ABB RobotStudio station: Cell1234 280921_GPA546_A0610_publ2.rspag

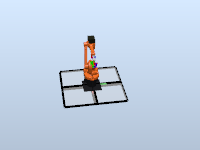
--- station ---
Station Cell1234 pubV2 (saved by RobotStudio 21.2.9526.0)
Controller 05-500633_Cell1, task T_PRINCIP: task frame (RAPID world) sits at (0, 0, 393.01) mm in the station
Controller 05-500633_Cell1
  mechanical unit ROB_1: IRB1600_5_145__01_2, 6 joints, base frame (0, 0, 0) mm
Layout (positions relative to the parent item):
  - Pince [mechanism, from Libraries\Pince.rslib] at (451.32, -3.6, 1437.47) mm, rotated rx 176.02 ry -40.72 rz 6.49 deg; joint values [0.0086] (rad or m)
  - BaseRobot [part, from Libraries\BaseRobot.rslib] at (0, 0, 38.61) mm, rotated rx 90 ry 0 rz 90 deg
  - BoitePince [part, from Libraries\BoitePince.rslib] at (-322.09, -37.25, -99.49) mm, rotated rx 0.01 ry 0.17 rz 1.48 deg
  - LogicGate [smart component, from Libraries\LogicGate.rslib]
      properties: Operator=AND; Delay=0
  - LogicGate [smart component, from Libraries\LogicGate.rslib]
      properties: Operator=NOT; Delay=0
  - IRB1600_5_145__01_2 [mechanism, from Robots\IRB1600_5_145__01.rslib] at (0, 0, 393.01) mm; joint values [-0.0095, -0.5091, 0.516, 0.0144, 0.8505, -1.6733] (rad or m)
  - Cellule_1_Composantes [graphiccomponentgroup]
    - 1_Bloc1 [part, from Libraries\Bloc1.rslib] at (-359.6, 653.4, 807.5) mm, rotated rx 126 ry 0 rz 95.5 deg
    - 1_Bloc2 [part, from Libraries\Bloc1.rslib] at (-359.6, 653.4, 807.5) mm, rotated rx 126 ry 0 rz 95.5 deg
    - 1_Bloc3 [part, from Libraries\Bloc3.rslib] at (-359.6, 653.4, 807.5) mm, rotated rx 126 ry 0 rz 95.5 deg
    - 1_Bloc4 [part, from Libraries\Bloc1.rslib] at (-359.6, 653.4, 807.5) mm, rotated rx 126 ry 0 rz 95.5 deg
    - 1_Bloc5 [part, from Libraries\Bloc1.rslib] at (-359.6, 653.4, 807.5) mm, rotated rx 126 ry 0 rz 95.5 deg
    - 1_Bloc6 [part, from Libraries\Bloc1.rslib] at (-359.6, 653.4, 807.5) mm, rotated rx 126 ry 0 rz 95.5 deg
    - 1_Bloc7 [part, from Libraries\Bloc1.rslib] at (-359.6, 653.4, 807.5) mm, rotated rx 126 ry 0 rz 95.5 deg
    - 1_Bloc8 [part, from Libraries\Bloc1.rslib] at (-359.6, 653.4, 807.5) mm, rotated rx 126 ry 0 rz 95.5 deg
    - 1_Bloc9 [part, from Libraries\Bloc1.rslib] at (-359.6, 653.4, 807.5) mm, rotated rx 126 ry 0 rz 95.5 deg
    - 1_Bloc10 [part, from Libraries\Bloc1.rslib] at (-359.6, 653.4, 807.5) mm, rotated rx 126 ry 0 rz 95.5 deg
    - 1_Crayon [part, from Libraries\Crayon.rslib] at (-244.5, 1025, 746) mm, rotated rx 180 ry 0 rz 0 deg
    - 1_Feuille8.5x11 [part, from Libraries\Feuille8.5x11.rslib] at (50, 800, 746.18) mm, rotated rx 0 ry 0 rz 30 deg
    - 1_Glissoire [part, from Libraries\Glissoire.rslib] at (-578.28, 671.48, 751.2) mm, rotated rx 0 ry 0 rz 5.91 deg
    - 1_PorteCrayon [part, from Libraries\PorteCrayon.rslib] at (-244.76, 1025.26, 745.91) mm
    - 1_Table [part, from Libraries\Table.rslib] at (-567.99, 565.9, -5.81) mm, rotated rx 0 ry 0 rz 5.91 deg
    - 1_Piston [mechanism, from Libraries\Piston.rslib] at (-578.34, 672.08, 752) mm, rotated rx 0 ry 0 rz 5.91 deg; joint values [0] (rad or m)
  - Cellule_2_Composantes [graphiccomponentgroup] at (0, 0, 0) mm
    - 2_Crayon [part, from Libraries\Crayon.rslib] at (-467.39, -707.37, 733.8) mm, rotated rx 179.84 ry -1.57 rz -98.83 deg
    - 2_Feuille8.5x11 [part, from Libraries\Feuille8.5x11.rslib] at (-232.98, -884.29, 745.95) mm, rotated rx -0.47 ry -0.18 rz -45.11 deg
    - 2_PorteCrayon [part, from Libraries\PorteCrayon.rslib] at (-467.32, -707.23, 738.97) mm, rotated rx -0.13 ry -1.57 rz -98.83 deg
    - 2_Table [part, from Libraries\Table.rslib] at (-872.9, -1097.81, -9.38) mm, rotated rx -0.48 ry 0.14 rz -7.29 deg
    - 2_Piston [mechanism, from Libraries\Piston.rslib] at (-862.29, -990.75, 748.42) mm, rotated rx -0.48 ry 0.15 rz -6.57 deg; joint values [0] (rad or m)
    - 2_Bloc1 [part, from Libraries\Bloc1.rslib] at (-652.89, -1053.85, 803.97) mm, rotated rx 126.28 ry 0.71 rz 83.59 deg
    - 2_Bloc2 [part, from Libraries\Bloc1.rslib] at (-652.89, -1053.85, 803.97) mm, rotated rx 126.28 ry 0.71 rz 83.89 deg
    - 2_Bloc3 [part, from Libraries\Bloc3.rslib] at (-652.89, -1053.85, 803.97) mm, rotated rx 126.28 ry 0.71 rz 83.59 deg
    - 2_Bloc4 [part, from Libraries\Bloc1.rslib] at (-652.89, -1053.85, 803.97) mm, rotated rx 126.28 ry 0.71 rz 83.59 deg
    - 2_Bloc5 [part, from Libraries\Bloc1.rslib] at (-652.89, -1053.85, 803.97) mm, rotated rx 126.28 ry 0.71 rz 83.59 deg
    - 2_Bloc6 [part, from Libraries\Bloc1.rslib] at (-652.89, -1053.85, 803.97) mm, rotated rx 126.28 ry 0.71 rz 83.59 deg
    - 2_Bloc7 [part, from Libraries\Bloc1.rslib] at (-652.89, -1053.85, 803.97) mm, rotated rx 126.28 ry 0.71 rz 83.59 deg
    - 2_Bloc8 [part, from Libraries\Bloc1.rslib] at (-652.89, -1053.85, 803.97) mm, rotated rx 126.28 ry 0.71 rz 83.59 deg
    - 2_Bloc9 [part, from Libraries\Bloc1.rslib] at (-652.89, -1053.85, 803.97) mm, rotated rx 126.28 ry 0.71 rz 83.59 deg
    - 2_Bloc10 [part, from Libraries\Bloc1.rslib] at (-652.89, -1053.85, 803.97) mm, rotated rx 126.28 ry 0.71 rz 83.59 deg
    - 2_Glissoire [part, from Libraries\Glissoire.rslib] at (-862.4, -991.66, 747.63) mm, rotated rx -0.48 ry 0.15 rz -6.57 deg
  - Cellule_4_Composantes [graphiccomponentgroup]
    - 4_Bloc1 [part, from Libraries\Bloc1.rslib] at (63.43, -1118.07, 750.5) mm, rotated rx 125.72 ry -2.22 rz 111.85 deg
    - 4_Bloc2 [part, from Libraries\Bloc1.rslib] at (63.43, -1118.07, 750.5) mm, rotated rx 125.72 ry -2.22 rz 111.85 deg
    - 4_Bloc3 [part, from Libraries\Bloc3.rslib] at (63.43, -1118.07, 750.5) mm, rotated rx 125.72 ry -2.22 rz 111.85 deg
    - 4_Bloc4 [part, from Libraries\Bloc1.rslib] at (63.43, -1118.07, 750.5) mm, rotated rx 125.72 ry -2.22 rz 111.85 deg
    - 4_Bloc5 [part, from Libraries\Bloc1.rslib] at (63.43, -1118.07, 750.5) mm, rotated rx 125.72 ry -2.22 rz 111.85 deg
    - 4_Bloc6 [part, from Libraries\Bloc1.rslib] at (63.43, -1118.07, 750.5) mm, rotated rx 125.72 ry -2.22 rz 111.85 deg
    - 4_Bloc7 [part, from Libraries\Bloc1.rslib] at (63.43, -1118.07, 750.5) mm, rotated rx 125.72 ry -2.22 rz 111.85 deg
    - 4_Bloc8 [part, from Libraries\Bloc1.rslib] at (63.43, -1118.07, 750.5) mm, rotated rx 125.72 ry -2.22 rz 111.85 deg
    - 4_Bloc9 [part, from Libraries\Bloc1.rslib] at (63.43, -1118.07, 750.5) mm, rotated rx 125.72 ry -2.22 rz 111.85 deg
    - 4_Bloc10 [part, from Libraries\Bloc1.rslib] at (63.43, -1118.07, 750.5) mm, rotated rx 125.72 ry -2.22 rz 111.85 deg
    - 4_Crayon [part, from Libraries\Crayon.rslib] at (94.76, -713.92, 704.73) mm, rotated rx 177.67 ry 0.01 rz -158.51 deg
    - 4_Feuille8.5x11 [part, from Libraries\Feuille8.5x11.rslib] at (445.38, -893.28, 690.04) mm, rotated rx 2.33 ry -0.01 rz 21.49 deg
    - 4_PorteCrayon [part, from Libraries\PorteCrayon.rslib] at (94.76, -713.92, 704.73) mm, rotated rx 2.33 ry -0.01 rz 21.49 deg
    - 4_Glissoire [part, from Libraries\Glissoire.rslib] at (-151.57, -1158.7, 694.69) mm, rotated rx 2.33 ry -0.01 rz 21.49 deg
    - 4_Table [part, from Libraries\Table.rslib] at (-113.25, -1225.41, -65.44) mm, rotated rx 2.33 ry -0.01 rz 21.49 deg
    - 4_Piston [mechanism, from Libraries\Piston.rslib] at (-151.91, -1157.85, 695.52) mm, rotated rx 2.33 ry -0.01 rz 21.49 deg; joint values [0] (rad or m)
  - Cellule_3_Composantes [graphiccomponentgroup]
    - 3_Bloc1 [part, from Libraries\Bloc1.rslib] at (-255.93, 676.35, 796.95) mm, rotated rx 125.68 ry -0.79 rz 86.11 deg
    - 3_Bloc2 [part, from Libraries\Bloc1.rslib] at (-255.93, 676.35, 796.95) mm, rotated rx 125.68 ry -0.79 rz 86.11 deg
    - 3_Bloc3 [part, from Libraries\Bloc3.rslib] at (-255.93, 676.35, 796.95) mm, rotated rx 125.68 ry -0.79 rz 86.11 deg
    - 3_Bloc4 [part, from Libraries\Bloc1.rslib] at (-255.93, 676.35, 796.95) mm, rotated rx 125.68 ry -0.79 rz 86.11 deg
    - 3_Bloc5 [part, from Libraries\Bloc1.rslib] at (-255.93, 676.35, 796.95) mm, rotated rx 125.68 ry -0.79 rz 86.11 deg
    - 3_Bloc6 [part, from Libraries\Bloc1.rslib] at (-255.93, 676.35, 796.95) mm, rotated rx 125.68 ry -0.79 rz 86.11 deg
    - 3_Bloc7 [part, from Libraries\Bloc1.rslib] at (-255.93, 676.35, 796.95) mm, rotated rx 125.68 ry -0.79 rz 86.11 deg
    - 3_Bloc8 [part, from Libraries\Bloc1.rslib] at (-255.93, 676.35, 796.95) mm, rotated rx 125.68 ry -0.79 rz 86.11 deg
    - 3_Bloc9 [part, from Libraries\Bloc1.rslib] at (-255.93, 676.35, 796.95) mm, rotated rx 126.68 ry -0.79 rz 86.11 deg
    - 3_Bloc10 [part, from Libraries\Bloc1.rslib] at (-255.93, 676.35, 796.95) mm, rotated rx 125.68 ry -0.79 rz 86.11 deg
    - 3_Crayon [part, from Libraries\Crayon.rslib] at (-66.31, 1010.69, 738.78) mm, rotated rx -179.88 ry 1.4 rz -95.14 deg
    - 3_Feuille8.5x11 [part, from Libraries\Feuille8.5x11.rslib] at (52.4, 669.01, 746.18) mm, rotated rx 0 ry 0 rz 1.76 deg
    - 3_Glissoire [part, from Libraries\Glissoire.rslib] at (-467.56, 729.54, 741.03) mm, rotated rx 0.36 ry 0.24 rz -3.84 deg
    - 3_PorteCrayon [part, from Libraries\PorteCrayon.rslib] at (-66.84, 1007.76, 860.12) mm, rotated rx -179.88 ry 1.4 rz -95.14 deg
    - 3_Table [part, from Libraries\Table.rslib] at (-484.28, 629.79, -18.55) mm, rotated rx 0.28 ry 0 rz -5.2 deg
    - 3_Piston [mechanism, from Libraries\Piston.rslib] at (-467.45, 731.2, 741.83) mm, rotated rx 0.36 ry 0.24 rz -3.84 deg; joint values [0] (rad or m)
Attachment: 1_PorteCrayon is attached to 1_Table
Attachment: 1_Piston is attached to 1_Glissoire
Attachment: Pince is attached to IRB1600_5_145__01_2 / Link6
Attachment: BoitePince is attached to IRB1600_5_145__01_2 / Link3
Attachment: 2_PorteCrayon is attached to 2_Table
Attachment: 2_Piston is attached to 2_Glissoire
Attachment: 4_PorteCrayon is attached to 4_Table
Attachment: 4_Piston is attached to 4_Glissoire
Attachment: 3_PorteCrayon is attached to 3_Table
Attachment: 3_Piston is attached to 3_Glissoire
EventTableEntry 2774: Group=, Trigger=DO01_EE_PINCE01 2775, Actions=[EventTableActionAttach 2776], Comment=Attache l'objet le plus proche a la pince, devrait normalement être un bloc quand dans le glissoire ou le crayon, ActivationMode=2, Cyclic=false
EventTableTriggerIO 2775: IOValue=[1], IRC5Controller=? -1, Operator=0, SignalSource=05-500633_Cell1 2885
EventTableActionAttach 2776: AttachmentParent=Pince 925, AttachmentChild=? -1, MountObject=false, Offset=[X=1, Y=0, Z=0, W=0, X=0, Y=1, Z=0, W=0, X=0, Y=0, Z=1, W=0, X=0, Y=0, Z=0, W=1], FlangeIndext=0, FindNearest=true
EventTableTriggerIO 2777: IOValue=[0], IRC5Controller=? -1, Operator=0, SignalSource=05-500633_Cell1 2885
EventTableEntry 2778: Group=, Trigger=DO01_EE_PINCE01 2777, Actions=[EventTableActionDetach 2779], Comment=relache ce que le robot tiens., ActivationMode=2, Cyclic=false
EventTableActionDetach 2779: AttachmentParent=Pince 925, AttachmentChild=? -1
EventTableEntry 2780: Group=, Trigger=INIT_GAUCHE 2781, Actions=[EventTableActionMove 5190, EventTableActionMove 5191, EventTableActionMove 5192, EventTableActionMove 5193, EventTableActionMove 5194, EventTableActionMove 5195, EventTableActionMove 5196, EventTableActionMove 5197, EventTableActionMove 5198, EventTableActionMove 5199, EventTableActionMove 5200, EventTableActionMove 5201, EventTableActionMove 5202, EventTableActionMove 5203, EventTableActionMove 5204, EventTableActionDetach 5205, DO09_FV0101 5206, PistonIN 5207, PistonOUT 5208, DI13_ZS0103 5209, DI09_ZS0101 5210, TrouAGauche 5211, INIT_GAUCHE 5212, INIT_DROITE 5213, EventTableActionMove 5214, EventTableActionMove 5215, EventTableActionMove 5216, EventTableActionMove 5217, EventTableActionMove 5218, EventTableActionMove 5219, EventTableActionMove 5220, EventTableActionMove 5221, EventTableActionMove 5222, EventTableActionMove 5223, EventTableActionMove 5237, EventTableActionMove 5238, EventTableActionMove 5239, EventTableActionMove 5240, EventTableActionMove 5241, EventTableActionMove 5242, EventTableActionMove 5243, EventTableActionMove 5244, EventTableActionMove 5245, EventTableActionMove 5246, EventTableActionMove 5247, EventTableActionMove 5248, EventTableActionMove 5249, EventTableActionMove 5250, EventTableActionMove 5251, EventTableActionMove 5252, EventTableActionMove 5253, EventTableActionMove 5254, EventTableActionMove 5255, EventTableActionMove 5256], Comment=Replace les 10 blocs dans la zone de prise,
replace le glissoire
replace la table
replace la feuille
replace le crayon et sa base
détache ce que la pince peut tenir
place les valeurs du verin, ActivationMode=2, Cyclic=false
EventTableTriggerIO 2781: IOValue=[1], IRC5Controller=? -1, Operator=0, SignalSource=Cell1234 pubV2 1
EventTableEntry 2812: Group=, Trigger=DO01_EE_PINCE01 2813, Actions=[EventTableActionMechanicalPose 2814], Comment=, ActivationMode=2, Cyclic=false
EventTableTriggerIO 2813: IOValue=[1], IRC5Controller=? -1, Operator=0, SignalSource=05-500633_Cell1 2885
EventTableActionMechanicalPose 2814: VirtualSignal=, Mechanism=Pince 925, ToPoseName=Closed, VirtualSignalValue=[1]
EventTableTriggerIO 2815: IOValue=[0], IRC5Controller=? -1, Operator=0, SignalSource=05-500633_Cell1 2885
EventTableEntry 2816: Group=, Trigger=DO01_EE_PINCE01 2815, Actions=[EventTableActionMechanicalPose 2817], Comment=, ActivationMode=2, Cyclic=false
EventTableActionMechanicalPose 2817: VirtualSignal=, Mechanism=Pince 925, ToPoseName=Opened, VirtualSignalValue=[1]
EventTableEntry 2818: Group=, Trigger=DO09_FV0101 2819, Actions=[EventTableActionMechanicalPose 2820, PistonIN 2822], Comment=, ActivationMode=2, Cyclic=false
EventTableTriggerIO 2819: IOValue=[1], IRC5Controller=? -1, Operator=0, SignalSource=05-500633_Cell1 2885
EventTableActionMechanicalPose 2820: VirtualSignal=PistonOUT, Mechanism=1_Piston 921, ToPoseName=OUT, VirtualSignalValue=[1]
EventTableTriggerIO 2821: IOValue=[0], IRC5Controller=? -1, Operator=0, SignalSource=05-500633_Cell1 2885
EventTableActionIO 2822: IOValue=[0], IRC5Controller=? -1, SignalTarget=Cell1234 pubV2 1
EventTableEntry 2823: Group=, Trigger=DO09_FV0101 2821, Actions=[EventTableActionMechanicalPose 2824, PistonOUT 2825], Comment=, ActivationMode=2, Cyclic=false
EventTableActionMechanicalPose 2824: VirtualSignal=PistonIN, Mechanism=1_Piston 921, ToPoseName=IN, VirtualSignalValue=[1]
EventTableActionIO 2825: IOValue=[0], IRC5Controller=? -1, SignalTarget=Cell1234 pubV2 1
EventTableTriggerIO 2847: IOValue=[1], IRC5Controller=? -1, Operator=0, SignalSource=Cell1234 pubV2 1
EventTableEntry 2848: Group=, Trigger=INIT_DROITE 2847, Actions=[EventTableActionMove 5156, EventTableActionMove 5157, EventTableActionMove 5158, EventTableActionMove 5159, EventTableActionMove 5160, EventTableActionMove 5161, EventTableActionMove 5162, EventTableActionMove 5163, EventTableActionMove 5164, EventTableActionMove 5165, EventTableActionMove 5166, EventTableActionMove 5167, EventTableActionMove 5168, EventTableActionMove 5169, EventTableActionMove 5170, EventTableActionDetach 5171, DO09_FV0101 5172, PistonIN 5173, PistonOUT 5174, DI13_ZS0103 5175, DI09_ZS0101 5176, TrouAGauche 5177, INIT_DROITE 5178, INIT_GAUCHE 5179, EventTableActionMove 5180, EventTableActionMove 5181, EventTableActionMove 5182, EventTableActionMove 5183, EventTableActionMove 5184, EventTableActionMove 5185, EventTableActionMove 5186, EventTableActionMove 5187, EventTableActionMove 5188, EventTableActionMove 5189, EventTableActionMove 5224, EventTableActionMove 5225, EventTableActionMove 5226, EventTableActionMove 5227, EventTableActionMove 5228, EventTableActionMove 5232, EventTableActionMove 5233, EventTableActionMove 5234, EventTableActionMove 5235, EventTableActionMove 5236, EventTableActionMove 5257, EventTableActionMove 5258, EventTableActionMove 5259, EventTableActionMove 5260, EventTableActionMove 5261, EventTableActionMove 5262, EventTableActionMove 5263, EventTableActionMove 5264, EventTableActionMove 5265, EventTableActionMove 5266], Comment=Replace les 10 blocs dans la zone de prise,
replace le glissoire
replace la table
replace la feuille
replace le crayon et sa base
détache ce que la pince peut tenir
place les valeurs du verin, ActivationMode=2, Cyclic=false
EventTableTriggerIO 3612: IOValue=[1], IRC5Controller=? -1, Operator=0, SignalSource=05-500633_Cell1 2885
EventTableTriggerIO 3613: IOValue=[0], IRC5Controller=? -1, Operator=0, SignalSource=05-500633_Cell1 2885
EventTableEntry 3614: Group=, Trigger=DO09_FV0101 3612, Actions=[EventTableActionMechanicalPose 3615, PistonIN 3616], Comment=, ActivationMode=2, Cyclic=false
EventTableActionMechanicalPose 3615: VirtualSignal=PistonOUT, Mechanism=2_Piston 3404, ToPoseName=OUT, VirtualSignalValue=[1]
EventTableActionIO 3616: IOValue=[0], IRC5Controller=? -1, SignalTarget=Cell1234 pubV2 1
EventTableEntry 3617: Group=, Trigger=DO09_FV0101 3613, Actions=[EventTableActionMechanicalPose 3618, PistonOUT 3619], Comment=, ActivationMode=2, Cyclic=false
EventTableActionMechanicalPose 3618: VirtualSignal=PistonIN, Mechanism=2_Piston 3404, ToPoseName=IN, VirtualSignalValue=[1]
EventTableActionIO 3619: IOValue=[0], IRC5Controller=? -1, SignalTarget=Cell1234 pubV2 1
EventTableTriggerIO 4329: IOValue=[1], IRC5Controller=? -1, Operator=0, SignalSource=05-500633_Cell1 2885
EventTableTriggerIO 4330: IOValue=[0], IRC5Controller=? -1, Operator=0, SignalSource=05-500633_Cell1 2885
EventTableEntry 4331: Group=, Trigger=DO09_FV0101 4329, Actions=[EventTableActionMechanicalPose 4332, PistonIN 4333], Comment=, ActivationMode=2, Cyclic=false
EventTableActionMechanicalPose 4332: VirtualSignal=PistonOUT, Mechanism=4_Piston 4323, ToPoseName=OUT, VirtualSignalValue=[1]
EventTableActionIO 4333: IOValue=[0], IRC5Controller=? -1, SignalTarget=Cell1234 pubV2 1
EventTableEntry 4334: Group=, Trigger=DO09_FV0101 4330, Actions=[EventTableActionMechanicalPose 4335, PistonOUT 4336], Comment=, ActivationMode=2, Cyclic=false
EventTableActionMechanicalPose 4335: VirtualSignal=PistonIN, Mechanism=4_Piston 4323, ToPoseName=IN, VirtualSignalValue=[1]
EventTableActionIO 4336: IOValue=[0], IRC5Controller=? -1, SignalTarget=Cell1234 pubV2 1
EventTableActionMove 5156: Object=1_Bloc1 943, GlobalTransform=[X=-0.095845752520224, Y=0.995396198367179, Z=0, W=0, X=0.585079205588221, Y=0.0563367198262618, Z=0.809016994374948, W=0, X=0.805292440615264, Y=0.0775408426275167, Z=-0.587785252292473, W=0, X=-0.3596, Y=0.6534, Z=0.8075, W=1]
EventTableActionMove 5157: Object=1_Bloc2 2784, GlobalTransform=[X=-0.095845752520224, Y=0.995396198367179, Z=0, W=0, X=0.585079205588221, Y=0.0563367198262618, Z=0.809016994374948, W=0, X=0.805292440615264, Y=0.0775408426275167, Z=-0.587785252292473, W=0, X=-0.3596, Y=0.6534, Z=0.8075, W=1]
EventTableActionMove 5158: Object=1_Bloc3 942, GlobalTransform=[X=-0.095845752520224, Y=0.995396198367179, Z=0, W=0, X=0.585079205588221, Y=0.0563367198262618, Z=0.809016994374948, W=0, X=0.805292440615264, Y=0.0775408426275167, Z=-0.587785252292473, W=0, X=-0.3596, Y=0.6534, Z=0.8075, W=1]
EventTableActionMove 5159: Object=1_Bloc4 2790, GlobalTransform=[X=-0.095845752520224, Y=0.995396198367179, Z=0, W=0, X=0.585079205588221, Y=0.0563367198262618, Z=0.809016994374948, W=0, X=0.805292440615264, Y=0.0775408426275167, Z=-0.587785252292473, W=0, X=-0.3596, Y=0.6534, Z=0.8075, W=1]
EventTableActionMove 5160: Object=1_Bloc5 2791, GlobalTransform=[X=-0.095845752520224, Y=0.995396198367179, Z=0, W=0, X=0.585079205588221, Y=0.0563367198262618, Z=0.809016994374948, W=0, X=0.805292440615264, Y=0.0775408426275167, Z=-0.587785252292473, W=0, X=-0.3596, Y=0.6534, Z=0.8075, W=1]
EventTableActionMove 5161: Object=1_Bloc6 2792, GlobalTransform=[X=-0.095845752520224, Y=0.995396198367179, Z=0, W=0, X=0.585079205588221, Y=0.0563367198262618, Z=0.809016994374948, W=0, X=0.805292440615264, Y=0.0775408426275167, Z=-0.587785252292473, W=0, X=-0.3596, Y=0.6534, Z=0.8075, W=1]
EventTableActionMove 5162: Object=1_Bloc7 2793, GlobalTransform=[X=-0.095845752520224, Y=0.995396198367179, Z=0, W=0, X=0.585079205588221, Y=0.0563367198262618, Z=0.809016994374948, W=0, X=0.805292440615264, Y=0.0775408426275167, Z=-0.587785252292473, W=0, X=-0.3596, Y=0.6534, Z=0.8075, W=1]
EventTableActionMove 5163: Object=1_Bloc8 2794, GlobalTransform=[X=-0.095845752520224, Y=0.995396198367179, Z=0, W=0, X=0.585079205588221, Y=0.0563367198262618, Z=0.809016994374948, W=0, X=0.805292440615264, Y=0.0775408426275167, Z=-0.587785252292473, W=0, X=-0.3596, Y=0.6534, Z=0.8075, W=1]
EventTableActionMove 5164: Object=1_Bloc9 2795, GlobalTransform=[X=-0.095845752520224, Y=0.995396198367179, Z=0, W=0, X=0.585079205588221, Y=0.0563367198262618, Z=0.809016994374948, W=0, X=0.805292440615264, Y=0.0775408426275167, Z=-0.587785252292473, W=0, X=-0.3596, Y=0.6534, Z=0.8075, W=1]
EventTableActionMove 5165: Object=1_Bloc10 2796, GlobalTransform=[X=-0.095845752520224, Y=0.995396198367179, Z=0, W=0, X=0.585079205588221, Y=0.0563367198262618, Z=0.809016994374948, W=0, X=0.805292440615264, Y=0.0775408426275167, Z=-0.587785252292473, W=0, X=-0.3596, Y=0.6534, Z=0.8075, W=1]
EventTableActionMove 5166: Object=1_Glissoire 932, GlobalTransform=[X=0.994684861284941, Y=0.102966143613121, Z=0, W=0, X=-0.102966143613121, Y=0.994684861284941, Z=0, W=0, X=0, Y=0, Z=1, W=0, X=-0.57828, Y=0.67148, Z=0.751202, W=1]
EventTableActionMove 5167: Object=1_Table 919, GlobalTransform=[X=0.994684861284941, Y=0.102966143613121, Z=0, W=0, X=-0.102966143613121, Y=0.994684861284941, Z=0, W=0, X=0, Y=0, Z=1, W=0, X=-0.567989, Y=0.565905, Z=-0.005814, W=1]
EventTableActionMove 5168: Object=1_Feuille8.5x11 933, GlobalTransform=[X=0.866025403784439, Y=0.5, Z=0, W=0, X=-0.5, Y=0.866025403784439, Z=0, W=0, X=0, Y=0, Z=1, W=0, X=0.05, Y=0.8, Z=0.746181, W=1]
EventTableActionMove 5169: Object=1_PorteCrayon 920, GlobalTransform=[X=1, Y=0, Z=0, W=0, X=0, Y=1, Z=0, W=0, X=0, Y=0, Z=1, W=0, X=-0.244763, Y=1.025263, Z=0.745911, W=1]
EventTableActionMove 5170: Object=1_Crayon 934, GlobalTransform=[X=1, Y=0, Z=0, W=0, X=0, Y=-1, Z=0, W=0, X=0, Y=0, Z=-1, W=0, X=-0.2445, Y=1.025, Z=0.746, W=1]
EventTableActionDetach 5171: AttachmentParent=Pince 925, AttachmentChild=? -1
EventTableActionIO 5172: IOValue=[0], IRC5Controller=? -1, SignalTarget=05-500633_Cell1 2885
EventTableActionIO 5173: IOValue=[1], IRC5Controller=? -1, SignalTarget=Cell1234 pubV2 1
EventTableActionIO 5174: IOValue=[0], IRC5Controller=? -1, SignalTarget=Cell1234 pubV2 1
EventTableActionIO 5175: IOValue=[1], IRC5Controller=? -1, SignalTarget=05-500633_Cell1 2885
EventTableActionIO 5176: IOValue=[1], IRC5Controller=? -1, SignalTarget=05-500633_Cell1 2885
EventTableActionIO 5177: IOValue=[0], IRC5Controller=? -1, SignalTarget=Cell1234 pubV2 1
EventTableActionIO 5178: IOValue=[0], IRC5Controller=? -1, SignalTarget=Cell1234 pubV2 1
EventTableActionIO 5179: IOValue=[0], IRC5Controller=? -1, SignalTarget=Cell1234 pubV2 1
EventTableActionMove 5180: Object=2_Bloc1 3408, GlobalTransform=[X=0.11163380406932, Y=0.993672151168342, Z=-0.0123915205480335, W=0, X=0.589147801205299, Y=-0.0561355574929458, Z=0.806072991434347, W=0, X=0.800276678483119, Y=-0.0972854314758168, Z=-0.591686388806258, W=0, X=-0.65289, Y=-1.05385, Z=0.80397, W=1]
EventTableActionMove 5181: Object=2_Bloc2 3409, GlobalTransform=[X=0.106429442376949, Y=0.994243040716826, Z=-0.0123915205480335, W=0, X=0.589433649061701, Y=-0.0530500314221419, Z=0.806072991434347, W=0, X=0.800775091488952, Y=-0.0930938781675272, Z=-0.591686388806258, W=0, X=-0.65289, Y=-1.05385, Z=0.80397, W=1]
EventTableActionMove 5182: Object=2_Bloc3 3410, GlobalTransform=[X=0.11163380406932, Y=0.993672151168342, Z=-0.0123915205480335, W=0, X=0.589147801205299, Y=-0.0561355574929458, Z=0.806072991434347, W=0, X=0.800276678483119, Y=-0.0972854314758168, Z=-0.591686388806258, W=0, X=-0.65289, Y=-1.05385, Z=0.80397, W=1]
EventTableActionMove 5183: Object=2_Bloc4 3411, GlobalTransform=[X=0.11163380406932, Y=0.993672151168342, Z=-0.0123915205480335, W=0, X=0.589147801205299, Y=-0.0561355574929458, Z=0.806072991434347, W=0, X=0.800276678483119, Y=-0.0972854314758168, Z=-0.591686388806258, W=0, X=-0.65289, Y=-1.05385, Z=0.80397, W=1]
EventTableActionMove 5184: Object=2_Bloc5 3412, GlobalTransform=[X=0.11163380406932, Y=0.993672151168342, Z=-0.0123915205480335, W=0, X=0.589147801205299, Y=-0.0561355574929458, Z=0.806072991434347, W=0, X=0.800276678483119, Y=-0.0972854314758168, Z=-0.591686388806258, W=0, X=-0.65289, Y=-1.05385, Z=0.80397, W=1]
EventTableActionMove 5185: Object=2_Bloc6 3413, GlobalTransform=[X=0.11163380406932, Y=0.993672151168342, Z=-0.0123915205480335, W=0, X=0.589147801205299, Y=-0.0561355574929458, Z=0.806072991434347, W=0, X=0.800276678483119, Y=-0.0972854314758168, Z=-0.591686388806258, W=0, X=-0.65289, Y=-1.05385, Z=0.80397, W=1]
EventTableActionMove 5186: Object=2_Bloc7 3414, GlobalTransform=[X=0.11163380406932, Y=0.993672151168342, Z=-0.0123915205480335, W=0, X=0.589147801205299, Y=-0.0561355574929458, Z=0.806072991434347, W=0, X=0.800276678483119, Y=-0.0972854314758168, Z=-0.591686388806258, W=0, X=-0.65289, Y=-1.05385, Z=0.80397, W=1]
EventTableActionMove 5187: Object=2_Bloc8 3415, GlobalTransform=[X=0.11163380406932, Y=0.993672151168342, Z=-0.0123915205480335, W=0, X=0.589147801205299, Y=-0.0561355574929458, Z=0.806072991434347, W=0, X=0.800276678483119, Y=-0.0972854314758168, Z=-0.591686388806258, W=0, X=-0.65289, Y=-1.05385, Z=0.80397, W=1]
EventTableActionMove 5188: Object=2_Bloc9 3416, GlobalTransform=[X=0.11163380406932, Y=0.993672151168342, Z=-0.0123915205480335, W=0, X=0.589147801205299, Y=-0.0561355574929458, Z=0.806072991434347, W=0, X=0.800276678483119, Y=-0.0972854314758168, Z=-0.591686388806258, W=0, X=-0.65289, Y=-1.05385, Z=0.80397, W=1]
EventTableActionMove 5189: Object=2_Bloc10 3417, GlobalTransform=[X=0.11163380406932, Y=0.993672151168342, Z=-0.0123915205480335, W=0, X=0.589147801205299, Y=-0.0561355574929458, Z=0.806072991434347, W=0, X=0.800276678483119, Y=-0.0972854314758168, Z=-0.591686388806258, W=0, X=-0.65289, Y=-1.05385, Z=0.80397, W=1]
EventTableActionMove 5190: Object=1_Bloc1 943, GlobalTransform=[X=0.0958457525202241, Y=-0.995396198367179, Z=0, W=0, X=-0.815380830769965, Y=-0.0785122441133584, Z=0.573576436351046, W=0, X=-0.570935804216825, Y=-0.0549748651699344, Z=-0.819152044288992, W=0, X=-0.3596, Y=0.6534, Z=0.8075, W=1]
EventTableActionMove 5191: Object=1_Bloc2 2784, GlobalTransform=[X=0.0958457525202241, Y=-0.995396198367179, Z=0, W=0, X=-0.815380830769965, Y=-0.0785122441133584, Z=0.573576436351046, W=0, X=-0.570935804216825, Y=-0.0549748651699344, Z=-0.819152044288992, W=0, X=-0.3596, Y=0.6534, Z=0.8075, W=1]
EventTableActionMove 5192: Object=1_Bloc3 942, GlobalTransform=[X=0.0958457525202241, Y=-0.995396198367179, Z=0, W=0, X=-0.815380830769965, Y=-0.0785122441133584, Z=0.573576436351046, W=0, X=-0.570935804216825, Y=-0.0549748651699344, Z=-0.819152044288992, W=0, X=-0.3596, Y=0.6534, Z=0.8075, W=1]
EventTableActionMove 5193: Object=1_Bloc4 2790, GlobalTransform=[X=0.0958457525202241, Y=-0.995396198367179, Z=0, W=0, X=-0.815380830769965, Y=-0.0785122441133584, Z=0.573576436351046, W=0, X=-0.570935804216825, Y=-0.0549748651699344, Z=-0.819152044288992, W=0, X=-0.3596, Y=0.6534, Z=0.8075, W=1]
EventTableActionMove 5194: Object=1_Bloc5 2791, GlobalTransform=[X=0.0958457525202241, Y=-0.995396198367179, Z=0, W=0, X=-0.815380830769965, Y=-0.0785122441133584, Z=0.573576436351046, W=0, X=-0.570935804216825, Y=-0.0549748651699344, Z=-0.819152044288992, W=0, X=-0.3596, Y=0.6534, Z=0.8075, W=1]
EventTableActionMove 5195: Object=1_Bloc6 2792, GlobalTransform=[X=0.0958457525202241, Y=-0.995396198367179, Z=0, W=0, X=-0.815380830769965, Y=-0.0785122441133584, Z=0.573576436351046, W=0, X=-0.570935804216825, Y=-0.0549748651699344, Z=-0.819152044288992, W=0, X=-0.3596, Y=0.6534, Z=0.8075, W=1]
EventTableActionMove 5196: Object=1_Bloc7 2793, GlobalTransform=[X=0.0958457525202241, Y=-0.995396198367179, Z=0, W=0, X=-0.815380830769965, Y=-0.0785122441133584, Z=0.573576436351046, W=0, X=-0.570935804216825, Y=-0.0549748651699344, Z=-0.819152044288992, W=0, X=-0.3596, Y=0.6534, Z=0.8075, W=1]
EventTableActionMove 5197: Object=1_Bloc8 2794, GlobalTransform=[X=0.0958457525202241, Y=-0.995396198367179, Z=0, W=0, X=-0.815380830769965, Y=-0.0785122441133584, Z=0.573576436351046, W=0, X=-0.570935804216825, Y=-0.0549748651699344, Z=-0.819152044288992, W=0, X=-0.3596, Y=0.6534, Z=0.8075, W=1]
EventTableActionMove 5198: Object=1_Bloc9 2795, GlobalTransform=[X=0.0958457525202241, Y=-0.995396198367179, Z=0, W=0, X=-0.815380830769965, Y=-0.0785122441133584, Z=0.573576436351046, W=0, X=-0.570935804216825, Y=-0.0549748651699344, Z=-0.819152044288992, W=0, X=-0.3596, Y=0.6534, Z=0.8075, W=1]
EventTableActionMove 5199: Object=1_Bloc10 2796, GlobalTransform=[X=0.0958457525202241, Y=-0.995396198367179, Z=0, W=0, X=-0.815380830769965, Y=-0.0785122441133584, Z=0.573576436351046, W=0, X=-0.570935804216825, Y=-0.0549748651699344, Z=-0.819152044288992, W=0, X=-0.3596, Y=0.6534, Z=0.8075, W=1]
EventTableActionMove 5200: Object=1_Glissoire 932, GlobalTransform=[X=0.994684861284941, Y=0.102966143613121, Z=0, W=0, X=-0.102966143613121, Y=0.994684861284941, Z=0, W=0, X=0, Y=0, Z=1, W=0, X=-0.57828, Y=0.67148, Z=0.751202, W=1]
EventTableActionMove 5201: Object=1_Table 919, GlobalTransform=[X=0.994684861284941, Y=0.102966143613121, Z=0, W=0, X=-0.102966143613121, Y=0.994684861284941, Z=0, W=0, X=0, Y=0, Z=1, W=0, X=-0.567989, Y=0.565905, Z=-0.005814, W=1]
EventTableActionMove 5202: Object=1_Feuille8.5x11 933, GlobalTransform=[X=0.866025403784439, Y=0.5, Z=0, W=0, X=-0.5, Y=0.866025403784439, Z=0, W=0, X=0, Y=0, Z=1, W=0, X=0.05, Y=0.8, Z=0.746181, W=1]
EventTableActionMove 5203: Object=1_PorteCrayon 920, GlobalTransform=[X=1, Y=0, Z=0, W=0, X=0, Y=1, Z=0, W=0, X=0, Y=0, Z=1, W=0, X=-0.244763, Y=1.025263, Z=0.745911, W=1]
EventTableActionMove 5204: Object=1_Crayon 934, GlobalTransform=[X=1, Y=0, Z=0, W=0, X=0, Y=-1, Z=0, W=0, X=0, Y=0, Z=-1, W=0, X=-0.2445, Y=1.025, Z=0.746, W=1]
EventTableActionDetach 5205: AttachmentParent=Pince 925, AttachmentChild=? -1
EventTableActionIO 5206: IOValue=[0], IRC5Controller=? -1, SignalTarget=05-500633_Cell1 2885
EventTableActionIO 5207: IOValue=[1], IRC5Controller=? -1, SignalTarget=Cell1234 pubV2 1
EventTableActionIO 5208: IOValue=[0], IRC5Controller=? -1, SignalTarget=Cell1234 pubV2 1
EventTableActionIO 5209: IOValue=[1], IRC5Controller=? -1, SignalTarget=05-500633_Cell1 2885
EventTableActionIO 5210: IOValue=[1], IRC5Controller=? -1, SignalTarget=05-500633_Cell1 2885
EventTableActionIO 5211: IOValue=[1], IRC5Controller=? -1, SignalTarget=Cell1234 pubV2 1
EventTableActionIO 5212: IOValue=[0], IRC5Controller=? -1, SignalTarget=Cell1234 pubV2 1
EventTableActionIO 5213: IOValue=[0], IRC5Controller=? -1, SignalTarget=Cell1234 pubV2 1
EventTableActionMove 5214: Object=2_Bloc1 3408, GlobalTransform=[X=-0.11163380406932, Y=-0.993672151168342, Z=0.0123915205480335, W=0, X=-0.589147801205299, Y=0.0561355574929458, Z=-0.806072991434347, W=0, X=0.800276678483119, Y=-0.0972854314758168, Z=-0.591686388806258, W=0, X=-0.65289, Y=-1.05385, Z=0.80397, W=1]
EventTableActionMove 5215: Object=2_Bloc2 3409, GlobalTransform=[X=-0.11163380406932, Y=-0.993672151168342, Z=0.0123915205480335, W=0, X=-0.589147801205299, Y=0.0561355574929458, Z=-0.806072991434347, W=0, X=0.800276678483119, Y=-0.0972854314758168, Z=-0.591686388806258, W=0, X=-0.65289, Y=-1.05385, Z=0.80397, W=1]
EventTableActionMove 5216: Object=2_Bloc3 3410, GlobalTransform=[X=-0.11163380406932, Y=-0.993672151168342, Z=0.0123915205480335, W=0, X=-0.589147801205299, Y=0.0561355574929458, Z=-0.806072991434347, W=0, X=0.800276678483119, Y=-0.0972854314758168, Z=-0.591686388806258, W=0, X=-0.65289, Y=-1.05385, Z=0.80397, W=1]
EventTableActionMove 5217: Object=2_Bloc4 3411, GlobalTransform=[X=-0.11163380406932, Y=-0.993672151168342, Z=0.0123915205480335, W=0, X=-0.589147801205299, Y=0.0561355574929458, Z=-0.806072991434347, W=0, X=0.800276678483119, Y=-0.0972854314758168, Z=-0.591686388806258, W=0, X=-0.65289, Y=-1.05385, Z=0.80397, W=1]
EventTableActionMove 5218: Object=2_Bloc5 3412, GlobalTransform=[X=-0.11163380406932, Y=-0.993672151168342, Z=0.0123915205480335, W=0, X=-0.589147801205299, Y=0.0561355574929458, Z=-0.806072991434347, W=0, X=0.800276678483119, Y=-0.0972854314758168, Z=-0.591686388806258, W=0, X=-0.65289, Y=-1.05385, Z=0.80397, W=1]
EventTableActionMove 5219: Object=2_Bloc7 3414, GlobalTransform=[X=-0.11163380406932, Y=-0.993672151168342, Z=0.0123915205480335, W=0, X=-0.589147801205299, Y=0.0561355574929458, Z=-0.806072991434347, W=0, X=0.800276678483119, Y=-0.0972854314758168, Z=-0.591686388806258, W=0, X=-0.65289, Y=-1.05385, Z=0.80397, W=1]
EventTableActionMove 5220: Object=2_Bloc8 3415, GlobalTransform=[X=-0.11163380406932, Y=-0.993672151168342, Z=0.0123915205480335, W=0, X=-0.590543649469635, Y=0.0563052670167674, Z=-0.805039076677186, W=0, X=0.799247203223194, Y=-0.0971873083208409, Z=-0.593092349673516, W=0, X=-0.65289, Y=-1.05385, Z=0.80397, W=1]
EventTableActionMove 5221: Object=2_Bloc9 3416, GlobalTransform=[X=-0.11163380406932, Y=-0.993672151168342, Z=0.0123915205480335, W=0, X=-0.589147801205299, Y=0.0561355574929458, Z=-0.806072991434347, W=0, X=0.800276678483119, Y=-0.0972854314758168, Z=-0.591686388806258, W=0, X=-0.65289, Y=-1.05385, Z=0.80397, W=1]
EventTableActionMove 5222: Object=2_Bloc10 3417, GlobalTransform=[X=-0.11163380406932, Y=-0.993672151168342, Z=0.0123915205480335, W=0, X=-0.589147801205299, Y=0.0561355574929458, Z=-0.806072991434347, W=0, X=0.800276678483119, Y=-0.0972854314758168, Z=-0.591686388806258, W=0, X=-0.65289, Y=-1.05385, Z=0.80397, W=1]
EventTableActionMove 5223: Object=2_Bloc6 3413, GlobalTransform=[X=-0.11163380406932, Y=-0.993672151168342, Z=0.0123915205480335, W=0, X=-0.589147801205299, Y=0.0561355574929458, Z=-0.806072991434347, W=0, X=0.800276678483119, Y=-0.0972854314758168, Z=-0.591686388806258, W=0, X=-0.65289, Y=-1.05385, Z=0.80397, W=1]
EventTableActionMove 5224: Object=3_Bloc1 4405, GlobalTransform=[X=0.0678347122764665, Y=0.997601299180121, Z=0.0137876642149455, W=0, X=0.581154167924004, Y=-0.0507426203388437, Z=0.81220996028472, W=0, X=0.810961333797689, Y=-0.047083270439542, Z=-0.583202263995768, W=0, X=-0.25593, Y=0.67635, Z=0.79695, W=1]
EventTableActionMove 5225: Object=3_Bloc2 4406, GlobalTransform=[X=0.0678347122764665, Y=0.997601299180121, Z=0.0137876642149455, W=0, X=0.581154167924004, Y=-0.0507426203388437, Z=0.81220996028472, W=0, X=0.810961333797689, Y=-0.047083270439542, Z=-0.583202263995768, W=0, X=-0.25593, Y=0.67635, Z=0.79695, W=1]
EventTableActionMove 5226: Object=3_Bloc3 4407, GlobalTransform=[X=0.0678347122764665, Y=0.997601299180121, Z=0.0137876642149455, W=0, X=0.581154167924004, Y=-0.0507426203388437, Z=0.81220996028472, W=0, X=0.810961333797689, Y=-0.047083270439542, Z=-0.583202263995768, W=0, X=-0.25593, Y=0.67635, Z=0.79695, W=1]
EventTableActionMove 5227: Object=3_Bloc4 4408, GlobalTransform=[X=0.0678347122764665, Y=0.997601299180121, Z=0.0137876642149455, W=0, X=0.581154167924004, Y=-0.0507426203388437, Z=0.81220996028472, W=0, X=0.810961333797689, Y=-0.047083270439542, Z=-0.583202263995768, W=0, X=-0.25593, Y=0.67635, Z=0.79695, W=1]
EventTableActionMove 5228: Object=3_Bloc5 4409, GlobalTransform=[X=0.0678347122764665, Y=0.997601299180121, Z=0.0137876642149455, W=0, X=0.581154167924004, Y=-0.0507426203388437, Z=0.81220996028472, W=0, X=0.810961333797689, Y=-0.047083270439542, Z=-0.583202263995768, W=0, X=-0.25593, Y=0.67635, Z=0.79695, W=1]
EventTableActionMove 5232: Object=3_Bloc6 4410, GlobalTransform=[X=0.0678347122764665, Y=0.997601299180121, Z=0.0137876642149455, W=0, X=0.581154167924004, Y=-0.0507426203388437, Z=0.81220996028472, W=0, X=0.810961333797689, Y=-0.047083270439542, Z=-0.583202263995768, W=0, X=-0.25593, Y=0.67635, Z=0.79695, W=1]
EventTableActionMove 5233: Object=3_Bloc7 4411, GlobalTransform=[X=0.0678347122764665, Y=0.997601299180121, Z=0.0137876642149455, W=0, X=0.581154167924004, Y=-0.0507426203388437, Z=0.81220996028472, W=0, X=0.810961333797689, Y=-0.047083270439542, Z=-0.583202263995768, W=0, X=-0.25593, Y=0.67635, Z=0.79695, W=1]
EventTableActionMove 5234: Object=3_Bloc8 4412, GlobalTransform=[X=0.0678347122764665, Y=0.997601299180121, Z=0.0137876642149455, W=0, X=0.581154167924004, Y=-0.0507426203388437, Z=0.81220996028472, W=0, X=0.810961333797689, Y=-0.047083270439542, Z=-0.583202263995768, W=0, X=-0.25593, Y=0.67635, Z=0.79695, W=1]
EventTableActionMove 5235: Object=3_Bloc9 4413, GlobalTransform=[X=0.0678347122764665, Y=0.997601299180121, Z=0.0137876642149455, W=0, X=0.595218882131705, Y=-0.0515566083640961, Z=0.801907973827343, W=0, X=0.800695281717241, Y=-0.0461905185955548, Z=-0.597288457805457, W=0, X=-0.25593, Y=0.67635, Z=0.79695, W=1]
EventTableActionMove 5236: Object=3_Bloc10 4414, GlobalTransform=[X=0.0678347122764665, Y=0.997601299180121, Z=0.0137876642149455, W=0, X=0.581154167924004, Y=-0.0507426203388437, Z=0.81220996028472, W=0, X=0.810961333797689, Y=-0.047083270439542, Z=-0.583202263995768, W=0, X=-0.25593, Y=0.67635, Z=0.79695, W=1]
EventTableActionMove 5237: Object=3_Bloc1 4405, GlobalTransform=[X=-0.0678347122764663, Y=-0.997601299180121, Z=-0.0137876642149455, W=0, X=0.581154167924004, Y=-0.0507426203388436, Z=0.81220996028472, W=0, X=-0.810961333797689, Y=0.0470832704395419, Z=0.583202263995768, W=0, X=-0.25593, Y=0.67635, Z=0.79695, W=1]
EventTableActionMove 5238: Object=3_Bloc2 4406, GlobalTransform=[X=-0.0678347122764663, Y=-0.997601299180121, Z=-0.0137876642149455, W=0, X=0.581154167924004, Y=-0.0507426203388436, Z=0.81220996028472, W=0, X=-0.810961333797689, Y=0.0470832704395419, Z=0.583202263995768, W=0, X=-0.25593, Y=0.67635, Z=0.79695, W=1]
EventTableActionMove 5239: Object=3_Bloc3 4407, GlobalTransform=[X=-0.0678347122764663, Y=-0.997601299180121, Z=-0.0137876642149455, W=0, X=0.581154167924004, Y=-0.0507426203388436, Z=0.81220996028472, W=0, X=-0.810961333797689, Y=0.0470832704395419, Z=0.583202263995768, W=0, X=-0.25593, Y=0.67635, Z=0.79695, W=1]
EventTableActionMove 5240: Object=3_Bloc4 4408, GlobalTransform=[X=-0.0678347122764663, Y=-0.997601299180121, Z=-0.0137876642149455, W=0, X=0.581154167924004, Y=-0.0507426203388436, Z=0.81220996028472, W=0, X=-0.810961333797689, Y=0.0470832704395419, Z=0.583202263995768, W=0, X=-0.25593, Y=0.67635, Z=0.79695, W=1]
EventTableActionMove 5241: Object=3_Bloc5 4409, GlobalTransform=[X=-0.0678347122764663, Y=-0.997601299180121, Z=-0.0137876642149455, W=0, X=0.581154167924004, Y=-0.0507426203388436, Z=0.81220996028472, W=0, X=-0.810961333797689, Y=0.0470832704395419, Z=0.583202263995768, W=0, X=-0.25593, Y=0.67635, Z=0.79695, W=1]
EventTableActionMove 5242: Object=3_Bloc6 4410, GlobalTransform=[X=-0.0678347122764663, Y=-0.997601299180121, Z=-0.0137876642149455, W=0, X=0.581154167924004, Y=-0.0507426203388436, Z=0.81220996028472, W=0, X=-0.810961333797689, Y=0.0470832704395419, Z=0.583202263995768, W=0, X=-0.25593, Y=0.67635, Z=0.79695, W=1]
EventTableActionMove 5243: Object=3_Bloc7 4411, GlobalTransform=[X=-0.0678347122764663, Y=-0.997601299180121, Z=-0.0137876642149455, W=0, X=0.581154167924004, Y=-0.0507426203388436, Z=0.81220996028472, W=0, X=-0.810961333797689, Y=0.0470832704395419, Z=0.583202263995768, W=0, X=-0.25593, Y=0.67635, Z=0.79695, W=1]
EventTableActionMove 5244: Object=3_Bloc8 4412, GlobalTransform=[X=-0.0678347122764663, Y=-0.997601299180121, Z=-0.0137876642149455, W=0, X=0.581154167924004, Y=-0.0507426203388436, Z=0.81220996028472, W=0, X=-0.810961333797689, Y=0.0470832704395419, Z=0.583202263995768, W=0, X=-0.25593, Y=0.67635, Z=0.79695, W=1]
EventTableActionMove 5245: Object=3_Bloc9 4413, GlobalTransform=[X=-0.0678347122764663, Y=-0.997601299180121, Z=-0.0137876642149455, W=0, X=0.581154167924004, Y=-0.0507426203388436, Z=0.81220996028472, W=0, X=-0.810961333797689, Y=0.0470832704395419, Z=0.583202263995768, W=0, X=-0.25593, Y=0.67635, Z=0.79695, W=1]
EventTableActionMove 5246: Object=3_Bloc10 4414, GlobalTransform=[X=-0.0678347122764663, Y=-0.997601299180121, Z=-0.0137876642149455, W=0, X=0.581154167924004, Y=-0.0507426203388436, Z=0.81220996028472, W=0, X=-0.810961333797689, Y=0.0470832704395419, Z=0.583202263995768, W=0, X=-0.25593, Y=0.67635, Z=0.79695, W=1]
EventTableActionMove 5247: Object=4_Bloc1 4308, GlobalTransform=[X=0.371898614723104, Y=-0.927464767525984, Z=-0.0387366153014063, W=0, X=0.553588298660916, Y=0.188096472128246, Z=0.811270431335089, W=0, X=-0.745138521318519, Y=-0.323154486539922, Z=0.583386460141449, W=0, X=0.06343, Y=-1.11807, Z=0.7505, W=1]
EventTableActionMove 5248: Object=4_Bloc2 4309, GlobalTransform=[X=0.371898614723104, Y=-0.927464767525984, Z=-0.0387366153014063, W=0, X=0.553588298660916, Y=0.188096472128246, Z=0.811270431335089, W=0, X=-0.745138521318519, Y=-0.323154486539922, Z=0.583386460141449, W=0, X=0.06343, Y=-1.11807, Z=0.7505, W=1]
EventTableActionMove 5249: Object=4_Bloc3 4310, GlobalTransform=[X=0.371898614723104, Y=-0.927464767525984, Z=-0.0387366153014063, W=0, X=0.553588298660916, Y=0.188096472128246, Z=0.811270431335089, W=0, X=-0.745138521318519, Y=-0.323154486539922, Z=0.583386460141449, W=0, X=0.06343, Y=-1.11807, Z=0.7505, W=1]
EventTableActionMove 5250: Object=4_Bloc4 4311, GlobalTransform=[X=0.371898614723104, Y=-0.927464767525984, Z=-0.0387366153014063, W=0, X=0.553588298660916, Y=0.188096472128246, Z=0.811270431335089, W=0, X=-0.745138521318519, Y=-0.323154486539922, Z=0.583386460141449, W=0, X=0.06343, Y=-1.11807, Z=0.7505, W=1]
EventTableActionMove 5251: Object=4_Bloc5 4312, GlobalTransform=[X=0.371898614723104, Y=-0.927464767525984, Z=-0.0387366153014063, W=0, X=0.553588298660916, Y=0.188096472128246, Z=0.811270431335089, W=0, X=-0.745138521318519, Y=-0.323154486539922, Z=0.583386460141449, W=0, X=0.06343, Y=-1.11807, Z=0.7505, W=1]
EventTableActionMove 5252: Object=4_Bloc6 4313, GlobalTransform=[X=0.371898614723104, Y=-0.927464767525984, Z=-0.0387366153014063, W=0, X=0.553588298660916, Y=0.188096472128246, Z=0.811270431335089, W=0, X=-0.745138521318519, Y=-0.323154486539922, Z=0.583386460141449, W=0, X=0.06343, Y=-1.11807, Z=0.7505, W=1]
EventTableActionMove 5253: Object=4_Bloc7 4314, GlobalTransform=[X=0.371898614723104, Y=-0.927464767525984, Z=-0.0387366153014063, W=0, X=0.553588298660916, Y=0.188096472128246, Z=0.811270431335089, W=0, X=-0.745138521318519, Y=-0.323154486539922, Z=0.583386460141449, W=0, X=0.06343, Y=-1.11807, Z=0.7505, W=1]
EventTableActionMove 5254: Object=4_Bloc8 4315, GlobalTransform=[X=0.371898614723104, Y=-0.927464767525984, Z=-0.0387366153014063, W=0, X=0.553588298660916, Y=0.188096472128246, Z=0.811270431335089, W=0, X=-0.745138521318519, Y=-0.323154486539922, Z=0.583386460141449, W=0, X=0.06343, Y=-1.11807, Z=0.7505, W=1]
EventTableActionMove 5255: Object=4_Bloc9 4316, GlobalTransform=[X=0.371898614723104, Y=-0.927464767525984, Z=-0.0387366153014063, W=0, X=0.553588298660916, Y=0.188096472128246, Z=0.811270431335089, W=0, X=-0.745138521318519, Y=-0.323154486539922, Z=0.583386460141449, W=0, X=0.06343, Y=-1.11807, Z=0.7505, W=1]
EventTableActionMove 5256: Object=4_Bloc10 4317, GlobalTransform=[X=0.371898614723104, Y=-0.927464767525984, Z=-0.0387366153014063, W=0, X=0.553588298660916, Y=0.188096472128246, Z=0.811270431335089, W=0, X=-0.745138521318519, Y=-0.323154486539922, Z=0.583386460141449, W=0, X=0.06343, Y=-1.11807, Z=0.7505, W=1]
EventTableActionMove 5257: Object=4_Bloc1 4308, GlobalTransform=[X=-0.371898614723104, Y=0.927464767525984, Z=0.0387366153014063, W=0, X=0.553588298660916, Y=0.188096472128246, Z=0.811270431335089, W=0, X=0.745138521318519, Y=0.323154486539922, Z=-0.583386460141449, W=0, X=0.06343, Y=-1.11807, Z=0.7505, W=1]
EventTableActionMove 5258: Object=4_Bloc2 4309, GlobalTransform=[X=-0.371898614723104, Y=0.927464767525984, Z=0.0387366153014063, W=0, X=0.553588298660916, Y=0.188096472128246, Z=0.811270431335089, W=0, X=0.745138521318519, Y=0.323154486539922, Z=-0.583386460141449, W=0, X=0.06343, Y=-1.11807, Z=0.7505, W=1]
EventTableActionMove 5259: Object=4_Bloc3 4310, GlobalTransform=[X=-0.371898614723104, Y=0.927464767525984, Z=0.0387366153014063, W=0, X=0.553588298660916, Y=0.188096472128246, Z=0.811270431335089, W=0, X=0.745138521318519, Y=0.323154486539922, Z=-0.583386460141449, W=0, X=0.06343, Y=-1.11807, Z=0.7505, W=1]
EventTableActionMove 5260: Object=4_Bloc4 4311, GlobalTransform=[X=-0.371898614723104, Y=0.927464767525984, Z=0.0387366153014063, W=0, X=0.553588298660916, Y=0.188096472128246, Z=0.811270431335089, W=0, X=0.745138521318519, Y=0.323154486539922, Z=-0.583386460141449, W=0, X=0.06343, Y=-1.11807, Z=0.7505, W=1]
EventTableActionMove 5261: Object=4_Bloc5 4312, GlobalTransform=[X=-0.371898614723104, Y=0.927464767525984, Z=0.0387366153014063, W=0, X=0.553588298660916, Y=0.188096472128246, Z=0.811270431335089, W=0, X=0.745138521318519, Y=0.323154486539922, Z=-0.583386460141449, W=0, X=0.06343, Y=-1.11807, Z=0.7505, W=1]
EventTableActionMove 5262: Object=4_Bloc6 4313, GlobalTransform=[X=-0.371898614723104, Y=0.927464767525984, Z=0.0387366153014063, W=0, X=0.553588298660916, Y=0.188096472128246, Z=0.811270431335089, W=0, X=0.745138521318519, Y=0.323154486539922, Z=-0.583386460141449, W=0, X=0.06343, Y=-1.11807, Z=0.7505, W=1]
EventTableActionMove 5263: Object=4_Bloc7 4314, GlobalTransform=[X=-0.371898614723104, Y=0.927464767525984, Z=0.0387366153014063, W=0, X=0.553588298660916, Y=0.188096472128246, Z=0.811270431335089, W=0, X=0.745138521318519, Y=0.323154486539922, Z=-0.583386460141449, W=0, X=0.06343, Y=-1.11807, Z=0.7505, W=1]
EventTableActionMove 5264: Object=4_Bloc8 4315, GlobalTransform=[X=-0.371898614723104, Y=0.927464767525984, Z=0.0387366153014063, W=0, X=0.553588298660916, Y=0.188096472128246, Z=0.811270431335089, W=0, X=0.745138521318519, Y=0.323154486539922, Z=-0.583386460141449, W=0, X=0.06343, Y=-1.11807, Z=0.7505, W=1]
EventTableActionMove 5265: Object=4_Bloc9 4316, GlobalTransform=[X=-0.371898614723104, Y=0.927464767525984, Z=0.0387366153014063, W=0, X=0.553588298660916, Y=0.188096472128246, Z=0.811270431335089, W=0, X=0.745138521318519, Y=0.323154486539922, Z=-0.583386460141449, W=0, X=0.06343, Y=-1.11807, Z=0.7505, W=1]
EventTableActionMove 5266: Object=4_Bloc10 4317, GlobalTransform=[X=-0.371898614723104, Y=0.927464767525984, Z=0.0387366153014063, W=0, X=0.553588298660916, Y=0.188096472128246, Z=0.811270431335089, W=0, X=0.745138521318519, Y=0.323154486539922, Z=-0.583386460141449, W=0, X=0.06343, Y=-1.11807, Z=0.7505, W=1]
Station signals: DI PistonIN, DI PistonOUT, DI INIT_GAUCHE, DI INIT_DROITE, DI TrouAGauche
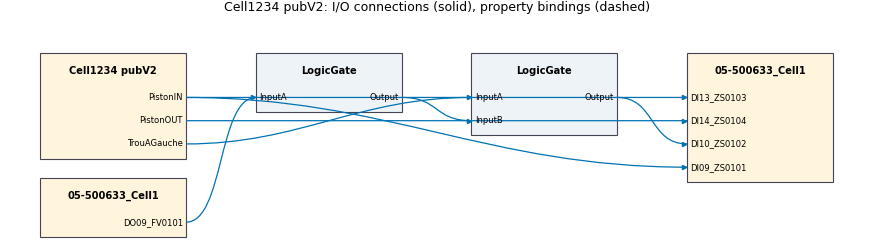
Station logic (signal -> signal, property => property):
  Cell1234 pubV2.PistonIN -> 05-500633_Cell1.DI13_ZS0103
  Cell1234 pubV2.PistonOUT -> 05-500633_Cell1.DI14_ZS0104
  Cell1234 pubV2.TrouAGauche -> LogicGate.InputA
  LogicGate.Output -> LogicGate.InputB
  LogicGate.Output -> 05-500633_Cell1.DI10_ZS0102
  05-500633_Cell1.DO09_FV0101 -> LogicGate.InputA
  Cell1234 pubV2.PistonIN -> 05-500633_Cell1.DI09_ZS0101
Targets, tools, work objects and paths stored in the station and not in the controller backup, written as RAPID:
! task T_PRINCIP
MODULE CalibData
  PERS tooldata MecanismePince_1:=[TRUE,[[0,0,226.245],[1,0,0,0]],[3,[0,0,100],[0,1,0,0],0,0,0]];
ENDMODULE

! task T_PRINCIP
MODULE CalibData
  PERS tooldata MecanismePince_1:=[TRUE,[[0,0,226.245],[1,0,0,0]],[3,[0,0,100],[0,1,0,0],0,0,0]];
  PERS tooldata Tooldata_1:=[TRUE,[[0,0,226.245],[1,0,0,0]],[3,[0,0,100],[0,1,0,0],0,0,0]];
ENDMODULE

! task T_PRINCIP
MODULE user
  PERS tooldata tPince_bout:=[TRUE,[[0,0,233.37],[0.707107,0,0,-0.707107]],[1.7,[12.2,0,158],[1,0,0,0],0.009,0.003,0.012]];
  PERS tooldata tSuce2:=[TRUE,[[38.1,42.545,222.174],[0.653281,-0.270598,-0.270598,-0.653281]],[1.7,[12.2,0,158],[1,0,0,0],0,0,0]];
  PERS tooldata tPince_bloc:=[TRUE,[[0,0,220],[0.707107,0,0,-0.707107]],[1.7,[12.2,0,158],[1,0,0,0],0.009,0.003,0.012]];
  PERS tooldata tCrayon:=[TRUE,[[0,0,283.37],[0.707107,0,0,-0.707107]],[1.7,[12.2,0,158],[1,0,0,0],0.009,0.003,0.012]];
  PERS tooldata tSuce1:=[TRUE,[[-38.1,42.545,222.174],[0.653281,-0.270598,-0.270598,-0.653281]],[1.7,[12.2,0,158],[1,0,0,0],0,0,0]];
  PERS tooldata tsuceCentre:=[TRUE,[[0,42.545,222.174],[0.653281,-0.270598,-0.270598,-0.653281]],[1.7,[12.2,0,158],[1,0,0,0],0,0,0]];
ENDMODULE


--- Backups/05-500633_Cell1/RAPID/TASK1/SYSMOD/LINKEDM.sys ---
%%%
  VERSION:1
  LANGUAGE:ENGLISH
%%%

MODULE LINKEDM (SYSMODULE)

! FOLLOWER
!     Name of electronically linked follower axis used by operator at teach pendent.
      PERS string l_f_axis_name{5}       :=  ["",  "", "", "", ""];

!     Name of the mechanical unit for follower axis.
      PERS string l_f_mecunt_n{5}  :=  ["", "", "", "", ""];

!     Linked follower axis number in the mechanical unit (first axis in mech. unit is number 1).
      PERS num l_f_axis_no{5}      :=  [0,          0,   0,  0,  0];

! MASTER
!     Name of the mechanical unit for linked master axis.
      PERS string l_m_mecunt_n{5} :=  ["", "", "", "", ""];

!     Linked master axis number in the mechanical unit (first axis in mech. unit is number 1).
!     See axis number table in documentation for different master mechanical units.
      PERS num l_m_axis_no{5}     :=  [0,  0,  0,  0,  0];

! POSITION OFFSET
!     The increase of the allowed offset position between the master and follower
!     positions, used when starting AUTO mode. As soon as the offset is decreased
!     the old configurated parameter is used.
!     Example: 3 => the configurated value of allowed offset is increased 3 times.
      PERS num offset_ratio{5}       :=  [10,  10,   10,  10,  10];

! SPEED RATIO
!     Speed_ratio used in AUTO and JOG modes [ very_slow   slow    normal    fast]
!     Value 1 = max allowed manual speed.
      CONST num speed_ratio {20}      := [0.01, 0.01, 0.01, 0.01, 0.01,
                                          0.05, 0.05, 0.05, 0.05, 0.05,
                                          0.20, 0.20, 0.20, 0.20, 0.20,
                                          1.00, 1.00, 1.00, 1.00, 1.00];

! STEP SIZE
!     Displacement position used in JOG mode for each activation of positive or
!     negative movement.                  [very_short    short   normal   long]
!     Unit degees or meter.
      CONST num displacement {20}     := [0.001, 0.001, 0.001, 0.001, 0.001,
                                          0.005, 0.005, 0.005, 0.005, 0.005,
                                          0.020, 0.020, 0.020, 0.020, 0.020,
                                          0.100, 0.100, 0.100, 0.100, 0.100];


!-------------------------------------------------------------
 PROC Linked_m ()
      Linked_m_exe ;
 ENDPROC
ENDMODULE

--- Backups/05-500633_Cell1/HOME/Lab1.mod ---
MODULE Lab1
! ----------------------------------------------------------------------------
! Programme : GPA546Lab1
! Auteurs : Mathieu Bélair, Raphael Archambault ET Simon Chaput
! Date : 1-18-18
! Révision : 0
!
! Description :
! Ce programme permet de prendre deux blocs dans une glissoire et de les
! superposer sur une table de travail.
! ----------------------------------------------------------------------------

  ! Donnees de type position enseignees
  PERS robtarget rGlissoire:=[[0,0,0],[1,0,0,0],[0,0,0,0],[9E+09,9E+09,9E+09,9E+09,9E+09,9E+09]];
  PERS robtarget rDepot:=[[0,0,0],[1,0,0,0],[0,0,0,0],[9E+09,9E+09,9E+09,9E+09,9E+09,9E+09]];
  PERS robtarget rRetrait:=[[0,0,0],[1,0,0,0],[0,0,0,0],[9E+09,9E+09,9E+09,9E+09,9E+09,9E+09]];

  ! Donnees de type position calculees
  VAR robtarget rDepot2;

  ! Donnees de type constante
  CONST num Epaisseur:=1; ! Épaisseur d'un bloc (en pouces)
  CONST num PouceToMM:=25.4; ! Facteur de conversion
  CONST num Decalage:=-200; ! Distance d'approche ou de retrait (mm)

  ! Données de type Variable
  VAR num EpaisMM:=0;

  ! Vitesse d'approche et de retrait (mm/sec)
  CONST speeddata LowSpeed:=[250,500,5000,1000];

  ! Vitesse maximale du robot (mm/sec)
  CONST speeddata HighSpeed:=[1000,500,5000,1000];

  ! Etat des entrees/sorties
  CONST dionum Ouverte:=0;
  CONST dionum Fermee:=1;
  CONST dionum Retracte:=0;
  CONST dionum Extension:=1;

  ! Variable pour limiter la zone de travail du robot
  VAR wztemporary EspaceRestreint;

! ----------------------------------------------------------------------------
! Procedure : main
! Auteurs : Yanick Noiseux
! Date : 4-08-2011
! Révision : 1.1
! Révision par: Martin Gaudreault
! Description :
! Routine qui est executee par le robot initialement.
! **** elle doit être en mode "cycle"
!
! ----------------------------------------------------------------------------
!**************************************************************************************
PROC main()

	! 1) Initialisation :
	init;

	! Deplacement a la position de repos
	MoveJ rRetrait, HighSpeed, fine, tPince_bloc\wobj:=wobj0;

	! 2) Calculs :
	EpaisMM := Epaisseur * PouceToMM; ! Conversion en mm
	rDepot2 := Offs(rDepot,0,0,EpaisMM);

	! 3) Déplacement du premier bloc :
	! Prise du bloc dans le glissoire
	Prise;
	! Dépôt du bloc 1 à la localisation rDepot :
	Depot(rDepot);

	! 4) Déplacement du deuxième bloc :
	! Prise du bloc dans le glissoire
	Prise;
	! Dépôt du bloc 2 à la localisation rDepot2 :
	Depot(rDepot2);

	! 5) Retourner le robot a la position de repos
	MoveJ rRetrait, HighSpeed, fine, tPince_bloc\wobj:=wobj0;

	Pince\Ouvert; ! Ouvrir la pince

ENDPROC
!**************************************************************************************

! ----------------------------------------------------------------------------
! Procedure : init
! Auteurs : Yanick Noiseux
! Date : 4-08-2011
! Révision : 1.1
! Révision par: Martin Gaudreault
! Description :
! Routine qui initialise les variables systèmes et les états des sorties
!
! ----------------------------------------------------------------------------
!**************************************************************************************
PROC init()

	! volume pour limiter les articulation du robot
	VAR shapedata joint_space;

	! Ne garder que les deux constantes correspondant a votre robot
	! Ces valeurs ne doivent pas être changées afin d'aider a la securite et représentent
    ! les limites logicielles pour chacun des axes

	! *** décommentez ces deux lignes si vous êtes sur le robot 1
	CONST jointtarget low_pos:=[[ 54, -25, -85, -90, -103, -289 ],[ 9E9, 9E9, 9E9, 9E9, 9E9, 9E9 ]];
	CONST jointtarget high_pos:=[[ 128,  55,  55,  90,  103,  109 ],[ 9E9, 9E9, 9E9, 9E9, 9E9, 9E9 ]];


	! activation de la limitation, obligatoire
	WZFree EspaceRestreint;
	WZLimJointDef \Outside, joint_space, low_pos, high_pos;
	WZLimSup \Temp, EspaceRestreint, joint_space;

	VelSet 25,1000; ! Limitation imposée pour la sécurité, obligatoire

	SetDO DO09_FV0101, Retracte; ! Rentrer le vérin
	Pince\Ouvert; ! Ouvrir la pince

ENDPROC
!**************************************************************************************

! ----------------------------------------------------------------------------
! Procedure : Prise
! Auteurs : Yanick Noiseux
! Date : 4-08-2011
! Révision : 1.0
!
! Description :
! Routine qui s'approche du glissoire, atends une piece,
! l'indexe et la prends de maniere securitaire
!
! ----------------------------------------------------------------------------
!**************************************************************************************
PROC Prise()

! Vérification de présence de bloc dans la glissoire
	IF DI09_ZS0101 = 0 THEN
		TPErase;
		TPWrite "Aucun bloc dans la glissoire";
		TPWrite "Placer deux bloc et remettre en mode AUTO";
		WaitDI DI09_ZS0101, 1; ! Attente d'un bloc
		Waittime 1; ! attente que le bloc se stabilise
	ENDIF

	! Prehension du bloc
	MoveJ RelTool(rGlissoire,0,0,Decalage),HighSpeed,z50,tPince_bloc\wobj:=wobj0;
	SetDO DO09_FV0101, Extension; ! Indexer le bloc durant le mouvement
	WAITDI DI14_ZS0104,1; ! Attendre pour le vérin sortie
	MoveL rGlissoire, LowSpeed, fine, tPince_bloc\wobj:=wobj0;
	Pince\Fermer; ! Fermer la pince
	SetDO DO09_FV0101, Retracte;
	WAITDI DI14_ZS0104,0;
	MoveL RelTool(rGlissoire,0,0,Decalage),LowSpeed,z50,tPince_bloc\wobj:=wobj0;

ENDPROC
!**************************************************************************************

! ----------------------------------------------------------------------------
! Procedure : Depot
! Auteurs : Yanick Noiseux
! Date : 4-08-2011
! Révision : 1.1
! Révision par: Martin Gaudreault
! Description :
! Routine qui initialise les variables systèmes et les états des sorties
!
! Parametre: recoit un robtarget où aller déposer le bloc avec aproche et degagement
!
! ----------------------------------------------------------------------------
!**************************************************************************************
PROC Depot(robtarget rPosDepot)

	MoveJ RelTool(rPosDepot,0,0,Decalage), HighSpeed, z50, tPince_bloc\wobj:=wobj0;
	MoveL rPosDepot, LowSpeed, fine, tPince_bloc;
	Pince\Ouvert; ! Ouvrir la pince
	MoveL RelTool(rPosDepot,0,0,Decalage), LowSpeed, z50, tPince_bloc\wobj:=wobj0;

ENDPROC
!**************************************************************************************

! ----------------------------------------------------------------------------
! Procedure : Pince
! Auteurs : Yanick Noiseux
! Date : 4-08-2011
! Révision : 1.1
! Révision par: Martin Gaudreault
! Description :
! Routine qui Défini l'état de l'outil pince du robot
! ----------------------------------------------------------------------------
!**************************************************************************************
PROC Pince(\switch Ouvert | switch Fermer)

    ! Action sur la pince
    IF Present(Fermer) THEN
		! verifie si la sortie doit-être changé d'état
		IF Doutput(DO01_EE_PINCE01)=0 THEN
       		Set DO01_EE_PINCE01; ! Ferme la pince
			WAITTIME 1;  !  Attente que la pince bouge physiquement
		ENDIF
    ELSE
		! verifie si la sortie doit-être changé d'état
		IF Doutput(DO01_EE_PINCE01)=1 THEN
       		Reset DO01_EE_PINCE01; ! Ferme la pince
			WAITTIME 1;  !  Attente que la pince bouge physiquement
		ENDIF
    ENDIF

ENDPROC
!**************************************************************************************
ENDMODULE

--- Backups/05-500633_Cell1/SYSPAR/EIO.cfg ---
EIO:CFG_1.0:6:1::
#
SYSSIG_OUT:

      -Status "MotorOn" -Signal "SDO_MON_MotorOn"

      -Status "MotorOff" -Signal "SDO_MON_MotorOff"

      -Status "CycleOn" -Signal "SDO_MON_CycleOn"

      -Status "EmStop" -Signal "SDO_MON_EStop"

      -Status "AutoOn" -Signal "SDO_MON_AutoOn"

      -Status "RunchOk" -Signal "SDO_MON_RunChainOK"

      -Status "Error" -Signal "SDO_MON_ExecError"

      -Status "MotOnState" -Signal "SDO_MON_MotorOnState"

      -Status "MotOffState" -Signal "SDO_MON_MotorOffState"

      -Status "MotSupTrigg" -Signal "SDO_MON_MotionSuprvTrig" -Arg1 "ROB_1"

      -Status "MotSupOn" -Signal "SDO_MON_MotionSuprvOn" -Arg1 "ROB_1"

      -Status "RegainDistError" -Signal "SDO_MON_PathReturnErr" -Arg1 "ROB_1"

      -Status "TaskExecuting" -Signal "SDO_MON_TaskExecMain" -Arg2 "T_PRINCIP"

      -Status "TCPSpeed" -Signal "SAO_MON_TCPSpeed" -Arg1 "ROB_1"
#
SYSSIG_IN:

      -Signal "SDI_ACT_MotorOn" -Action "MotorOn"

      -Signal "SDI_ACT_MotorOff" -Action "MotorOff"

      -Signal "SDI_ACT_StartAtCurrent_Cycle" -Action "Start" -Arg1 "CYCLE"

      -Signal "SDI_ACT_StartAtMain_Cycle" -Action "StartMain" -Arg1 "CYCLE"

      -Signal "SDI_ACT_Stop" -Action "Stop"

      -Signal "SDI_ACT_StopAtEndCycle" -Action "StopCycle"

      -Signal "SDI_ACT_ResetEStop" -Action "ResetEstop"

      -Signal "SDI_ACT_ResetExecError" -Action "ResetError"

      -Signal "SDI_ACT_StopAtEndInstr" -Action "StopInstr"

      -Signal "SDI_ACT_StartAtMain_Cont" -Action "StartMain" -Arg1 "CONT"

      -Signal "SDI_ACT_StartAtCurrent_Cont" -Action "Start" -Arg1 "CONT"
#
INDUSTRIAL_NETWORK:

      -Name "DeviceNet" -Label "DeviceNet Master/Slave Network" -Address "2"

      -Name "DeviceNet_Anybus" -Label "DeviceNet Anybus Network" -Address "8"
#
EIO_ACCESS:

      -Name "Local_AUTO" -Rapid  -LocalManual  -LocalAuto
#
DEVICENET_DEVICE:

      -Name "ModuleES_10" -VendorName "ABB Robotics"\
      -ProductName "24 VDC I/O Device" -Label "DSQC 652 24 VDC I/O Device"\
      -Address 10 -ProductCode 26 -DeviceType 7 -ConnectionType "COS"\
      -OutputSize 2 -InputSize 2

      -Name "Virtuel" -Simulated  -VendorName "ABB Robotics"\
      -ProductName "24 VDC I/O Device" -Label "DSQC 652 24 VDC I/O Device"\
      -ProductCode 26 -DeviceType 7 -ConnectionType "COS" -OutputSize 2\
      -InputSize 2
#
DEVICENET_INTERNAL_DEVICE:

      -Name "DN_Internal_Device" -VendorName "ABB Robotics"\
      -ProductName "DeviceNet Internal Slave Device"
#
DEVICENET_INTERNAL_ANYBUS_DEVICE:

      -Name "DNet_Slave" -VendorName "ABB Robotics"\
      -ProductName "DeviceNet Internal Anybus Slave Device" -OutputSize 24\
      -InputSize 24
#
EIO_SIGNAL:

      -Name "DI01_EE_VAC01" -SignalType "DI" -Device "ModuleES_10"\
      -Label "EE-Objet sur Ventouse 1" -DeviceMap "0" -Category "Effecteur"

      -Name "DI02_EE_VAC02" -SignalType "DI" -Device "ModuleES_10"\
      -Label "EE-Objet sur Ventouse 2" -DeviceMap "1" -Category "Effecteur"

      -Name "DO01_EE_PINCE01" -SignalType "DO" -Device "ModuleES_10"\
      -Label "EE-Pince 1, ACTION FERMETURE" -DeviceMap "0" -Category "Effecteur"

      -Name "DO02_EE_VENT01" -SignalType "DO" -Device "ModuleES_10"\
      -Label "EE-Ventouse 1, ACTION SUCCION" -DeviceMap "1"\
      -Category "Effecteur"

      -Name "DO03_EE_VENT02" -SignalType "DO" -Device "ModuleES_10"\
      -Label "EE-Ventouse 2, ACTION SUCCION" -DeviceMap "2"\
      -Category "Effecteur"

      -Name "DO04_EE_LampBlu" -SignalType "DO" -Device "ModuleES_10"\
      -Label "EE-Lampe bleue" -DeviceMap "3" -Category "Effecteur"

      -Name "DO05_EE_LampOr" -SignalType "DO" -Device "ModuleES_10"\
      -Label "EE-Lampe orange" -DeviceMap "4" -Category "Effecteur"

      -Name "DO09_FV0101" -SignalType "DO" -Device "ModuleES_10"\
      -Label "GLI-Vérin 1, ACTION EXTENSION" -DeviceMap "8"\
      -Category "Glissoire"

      -Name "DO06" -SignalType "DO" -Device "ModuleES_10"\
      -Label "DOUT06 (non utilisé)" -DeviceMap "5"

      -Name "DO07" -SignalType "DO" -Device "ModuleES_10"\
      -Label "DOUT07 (non utilisé)" -DeviceMap "6"

      -Name "DO08" -SignalType "DO" -Device "ModuleES_10"\
      -Label "DOUT08 (non utilisé)" -DeviceMap "7"

      -Name "DO10" -SignalType "DO" -Device "ModuleES_10"\
      -Label "DOUT10 (non utilisé)" -DeviceMap "9"

      -Name "DO11" -SignalType "DO" -Device "ModuleES_10"\
      -Label "DOUT11 (non utilisé)" -DeviceMap "10"

      -Name "DO12" -SignalType "DO" -Device "ModuleES_10"\
      -Label "DOUT12 (non utilisé)" -DeviceMap "11"

      -Name "DO13" -SignalType "DO" -Device "ModuleES_10"\
      -Label "DOUT13 (non utilisé)" -DeviceMap "12"

      -Name "DO14" -SignalType "DO" -Device "ModuleES_10"\
      -Label "DOUT14 (non utilisé)" -DeviceMap "13"

      -Name "DO16" -SignalType "DO" -Device "ModuleES_10"\
      -Label "DOUT16 (non utilisé)" -DeviceMap "15"

      -Name "DI03" -SignalType "DI" -Device "ModuleES_10"\
      -Label "DIN03 - Effecteur (non utilisé)" -DeviceMap "2"\
      -Category "Effecteur"

      -Name "DI05" -SignalType "DI" -Device "ModuleES_10"\
      -Label "DIN05 - Effecteur (non utilisé)" -DeviceMap "4"\
      -Category "Effecteur"

      -Name "DI04" -SignalType "DI" -Device "ModuleES_10"\
      -Label "DIN04 - Effecteur (non utilisé)" -DeviceMap "3"\
      -Category "Effecteur"

      -Name "DI06" -SignalType "DI" -Device "ModuleES_10"\
      -Label "DIN06, (non utilisé)" -DeviceMap "5"

      -Name "DI07" -SignalType "DI" -Device "ModuleES_10"\
      -Label "DIN07, (non utilisé)" -DeviceMap "6"

      -Name "DI08" -SignalType "DI" -Device "ModuleES_10"\
      -Label "DIN08, (non utilisé)" -DeviceMap "7"

      -Name "DI09_ZS0101" -SignalType "DI" -Device "ModuleES_10"\
      -Label "GLI-Bloc présent au poussoir" -DeviceMap "8" -Category "Glissoire"

      -Name "DI10_ZS0102" -SignalType "DI" -Device "ModuleES_10"\
      -Label "GLI-Bloc orienté" -DeviceMap "9" -Category "Glissoire"

      -Name "DI11_LSL0101" -SignalType "DI" -Device "ModuleES_10"\
      -Label "GLI-Bloc présent bas niveau" -DeviceMap "10" -Category "Glissoire"

      -Name "DI12_LSH0101" -SignalType "DI" -Device "ModuleES_10"\
      -Label "GLI-Bloc présent haut niveau" -DeviceMap "11"\
      -Category "Glissoire"

      -Name "DI13_ZS0103" -SignalType "DI" -Device "ModuleES_10"\
      -Label "GLI-Vérin position rétracté" -DeviceMap "12" -Category "Glissoire"

      -Name "DO15" -SignalType "DO" -Device "ModuleES_10"\
      -Label "DOUT15 (non utilisé)" -DeviceMap "14"

      -Name "DI14_ZS0104" -SignalType "DI" -Device "ModuleES_10"\
      -Label "GLI-Vérin position étendu" -DeviceMap "13" -Category "Glissoire"

      -Name "DI15" -SignalType "DI" -Device "ModuleES_10"\
      -Label "DIN15, (non utilisé)" -DeviceMap "14"

      -Name "DI16" -SignalType "DI" -Device "ModuleES_10"\
      -Label "DIN16, (non utilisé)" -DeviceMap "15"

      -Name "GrO_PLCIN_01" -SignalType "GO" -Device "DNet_Slave"\
      -Label "GrOUT 01/ 8 bit vers PLC " -DeviceMap "0-7" -Category "PLC"

      -Name "GrO_PLCIN_02" -SignalType "GO" -Device "DNet_Slave"\
      -Label "GrOUT 02/ 8 bit vers PLC " -DeviceMap "8-15" -Category "PLC"

      -Name "GrO_PLCIN_03" -SignalType "GO" -Device "DNet_Slave"\
      -Label "GrOUT 03/ 8 bit vers PLC " -DeviceMap "16-23" -Category "PLC"

      -Name "DO_PLCIN_00" -SignalType "DO" -Device "DNet_Slave"\
      -Label "DOUT vers PLC via DNET" -DeviceMap "32" -Category "PLC"

      -Name "DO_PLCIN_01" -SignalType "DO" -Device "DNet_Slave"\
      -Label "DOUT vers PLC via DNET" -DeviceMap "33" -Category "PLC"

      -Name "DO_PLCIN_02" -SignalType "DO" -Device "DNet_Slave"\
      -Label "DOUT vers PLC via DNET" -DeviceMap "34" -Category "PLC"

      -Name "DO_PLCIN_03" -SignalType "DO" -Device "DNet_Slave"\
      -Label "DOUT vers PLC via DNET" -DeviceMap "35" -Category "PLC"

      -Name "DO_PLCIN_04" -SignalType "DO" -Device "DNet_Slave"\
      -Label "DOUT vers PLC via DNET" -DeviceMap "36" -Category "PLC"

      -Name "DO_PLCIN_05" -SignalType "DO" -Device "DNet_Slave"\
      -Label "DOUT vers PLC via DNET" -DeviceMap "37" -Category "PLC"

      -Name "DO_PLCIN_06" -SignalType "DO" -Device "DNet_Slave"\
      -Label "DOUT vers PLC via DNET" -DeviceMap "38" -Category "PLC"

      -Name "DO_PLCIN_07" -SignalType "DO" -Device "DNet_Slave"\
      -Label "DOUT vers PLC via DNET" -DeviceMap "39" -Category "PLC"

      -Name "GrO_PLCIN_04" -SignalType "GO" -Device "DNet_Slave"\
      -Label "GrOUT 04/ 8 bit vers PLC " -DeviceMap "24-31" -Category "PLC"

      -Name "DI_PLCOUT_00" -SignalType "DI" -Device "DNet_Slave"\
      -Label "DIN du PLC via DNET" -DeviceMap "32" -Category "PLC"

      -Name "DI_PLCOUT_01" -SignalType "DI" -Device "DNet_Slave"\
      -Label "DIN du PLC via DNET" -DeviceMap "33" -Category "PLC"

      -Name "DI_PLCOUT_02" -SignalType "DI" -Device "DNet_Slave"\
      -Label "DIN du PLC via DNET" -DeviceMap "34" -Category "PLC"

      -Name "DI_PLCOUT_03" -SignalType "DI" -Device "DNet_Slave"\
      -Label "DIN du PLC via DNET" -DeviceMap "35" -Category "PLC"

      -Name "DI_PLCOUT_04" -SignalType "DI" -Device "DNet_Slave"\
      -Label "DIN du PLC via DNET" -DeviceMap "36" -Category "PLC"

      -Name "DI_PLCOUT_05" -SignalType "DI" -Device "DNet_Slave"\
      -Label "DIN du PLC via DNET" -DeviceMap "37" -Category "PLC"

      -Name "DI_PLCOUT_06" -SignalType "DI" -Device "DNet_Slave"\
      -Label "DIN du PLC via DNET" -DeviceMap "38" -Category "PLC"

      -Name "DI_PLCOUT_07" -SignalType "DI" -Device "DNet_Slave"\
      -Label "DIN du PLC via DNET" -DeviceMap "39" -Category "PLC"

      -Name "GrI_PLCOUT_01" -SignalType "GI" -Device "DNet_Slave"\
      -Label "GrOUT 01/ 8 bit vers PLC " -DeviceMap "0-7" -Category "PLC"

      -Name "GrI_PLCOUT_02" -SignalType "GI" -Device "DNet_Slave"\
      -Label "GrOUT 02/ 8 bit vers PLC " -DeviceMap "8-15" -Category "PLC"

      -Name "GrI_PLCOUT_03" -SignalType "GI" -Device "DNet_Slave"\
      -Label "GrOUT 03/ 8 bit vers PLC " -DeviceMap "16-23" -Category "PLC"

      -Name "GrI_PLCOUT_04" -SignalType "GI" -Device "DNet_Slave"\
      -Label "GrOUT 04/ 8 bit vers PLC " -DeviceMap "24-31" -Category "PLC"

      -Name "DI_PLCOUT_08" -SignalType "DI" -Device "DNet_Slave"\
      -Label "DIN du PLC via DNET" -DeviceMap "40" -Category "PLC"

      -Name "DI_PLCOUT_09" -SignalType "DI" -Device "DNet_Slave"\
      -Label "DIN du PLC via DNET" -DeviceMap "41" -Category "PLC"

      -Name "DI_PLCOUT_10" -SignalType "DI" -Device "DNet_Slave"\
      -Label "DIN du PLC via DNET" -DeviceMap "42" -Category "PLC"

      -Name "DI_PLCOUT_11" -SignalType "DI" -Device "DNet_Slave"\
      -Label "DIN du PLC via DNET" -DeviceMap "43" -Category "PLC"

      -Name "DI_PLCOUT_12" -SignalType "DI" -Device "DNet_Slave"\
      -Label "DIN du PLC via DNET" -DeviceMap "44" -Category "PLC"

      -Name "DI_PLCOUT_13" -SignalType "DI" -Device "DNet_Slave"\
      -Label "DIN du PLC via DNET" -DeviceMap "45" -Category "PLC"

      -Name "DI_PLCOUT_14" -SignalType "DI" -Device "DNet_Slave"\
      -Label "DIN du PLC via DNET" -DeviceMap "46" -Category "PLC"

      -Name "DI_PLCOUT_15" -SignalType "DI" -Device "DNet_Slave"\
      -Label "DIN du PLC via DNET" -DeviceMap "47" -Category "PLC"

      -Name "DO_PLCIN_08" -SignalType "DO" -Device "DNet_Slave"\
      -Label "DOUT vers PLC via DNET" -DeviceMap "40" -Category "PLC"

      -Name "DO_PLCIN_09" -SignalType "DO" -Device "DNet_Slave"\
      -Label "DOUT vers PLC via DNET" -DeviceMap "41" -Category "PLC"

      -Name "DO_PLCIN_10" -SignalType "DO" -Device "DNet_Slave"\
      -Label "DOUT vers PLC via DNET" -DeviceMap "42" -Category "PLC"

      -Name "DO_PLCIN_11" -SignalType "DO" -Device "DNet_Slave"\
      -Label "DOUT vers PLC via DNET" -DeviceMap "43" -Category "PLC"

      -Name "DO_PLCIN_12" -SignalType "DO" -Device "DNet_Slave"\
      -Label "DOUT vers PLC via DNET" -DeviceMap "44" -Category "PLC"

      -Name "DO_PLCIN_13" -SignalType "DO" -Device "DNet_Slave"\
      -Label "DOUT vers PLC via DNET" -DeviceMap "45" -Category "PLC"

      -Name "DO_PLCIN_14" -SignalType "DO" -Device "DNet_Slave"\
      -Label "DOUT vers PLC via DNET" -DeviceMap "46" -Category "PLC"

      -Name "DO_PLCIN_15" -SignalType "DO" -Device "DNet_Slave"\
      -Label "DOUT vers PLC via DNET" -DeviceMap "47" -Category "PLC"

      -Name "SDI_ACT_MotorOn" -SignalType "DI" -Device "DNet_Slave"\
      -Label "Activation moteurs SYSTEM IN du PLC" -DeviceMap "48"\
      -Category "PLC"

      -Name "SDI_ACT_MotorOff" -SignalType "DI" -Device "DNet_Slave"\
      -Label "Désactivation moteurs SYST IN du PLC" -DeviceMap "49"\
      -Category "PLC"

      -Name "SDI_ACT_StartAtCurrent_Cycle" -SignalType "DI" -Device "DNet_Slave"\
      -Label "Exec au PP mode Cycle SYSTEM IN du PLC" -DeviceMap "50"\
      -Category "PLC"

      -Name "SDI_ACT_StartAtMain_Cycle" -SignalType "DI" -Device "DNet_Slave"\
      -Label "Exec PP to Main mode Cycle SYSTEM IN du PLC" -DeviceMap "51"\
      -Category "PLC"

      -Name "SDI_ACT_Stop" -SignalType "DI" -Device "DNet_Slave"\
      -Label "Arrêt programme SYSTEM IN du PLC" -DeviceMap "52" -Category "PLC"

      -Name "SDI_ACT_StopAtEndCycle" -SignalType "DI" -Device "DNet_Slave"\
      -Label "Arrêt a la fin cycle SYSTEM IN du PLC" -DeviceMap "53"\
      -Category "PLC"

      -Name "SDI_ACT_ResetEStop" -SignalType "DI" -Device "DNet_Slave"\
      -Label "RAZ Arrêt urgence SYSTEM IN du PLC" -DeviceMap "54"\
      -Category "PLC"

      -Name "SDI_ACT_ResetExecError" -SignalType "DI" -Device "DNet_Slave"\
      -Label "RAZ Erreur exécution SYSTEM IN du PLC" -DeviceMap "55"\
      -Category "PLC"

      -Name "SDI_ACT_StopAtEndInstr" -SignalType "DI" -Device "DNet_Slave"\
      -Label "Arrêt a la fin instruction SYSTEM IN du PLC" -DeviceMap "56"\
      -Category "PLC"

      -Name "SDI_PLCOUT_11" -SignalType "DI" -Device "DNet_Slave"\
      -Label "SYSTEM IN du PLC via DNET" -DeviceMap "59" -Category "PLC"

      -Name "SDI_PLCOUT_12" -SignalType "DI" -Device "DNet_Slave"\
      -Label "SYSTEM IN du PLC via DNET" -DeviceMap "60" -Category "PLC"

      -Name "SDI_PLCOUT_13" -SignalType "DI" -Device "DNet_Slave"\
      -Label "SYSTEM IN du PLC via DNET" -DeviceMap "61" -Category "PLC"

      -Name "SDI_PLCOUT_14" -SignalType "DI" -Device "DNet_Slave"\
      -Label "SYSTEM IN du PLC via DNET" -DeviceMap "62" -Category "PLC"

      -Name "SDI_PLCOUT_15" -SignalType "DI" -Device "DNet_Slave"\
      -Label "SYSTEM IN du PLC via DNET" -DeviceMap "63" -Category "PLC"

      -Name "SDO_MON_MotorOn" -SignalType "DO" -Device "DNet_Slave"\
      -Label "Moteurs activés = 1, Non prêt = pulse SYSTEM OUT vers PLC"\
      -DeviceMap "48" -Category "PLC"

      -Name "SDO_MON_MotorOff" -SignalType "DO" -Device "DNet_Slave"\
      -Label "Moteurs désactivés = 1, Non prêt = pulse SYSTEM OUT vers PLC"\
      -DeviceMap "49" -Category "PLC"

      -Name "SDO_MON_CycleOn" -SignalType "DO" -Device "DNet_Slave"\
      -Label "Programme en exécution SYSTEM OUT vers PLC" -DeviceMap "50"\
      -Category "PLC"

      -Name "SDO_MON_EStop" -SignalType "DO" -Device "DNet_Slave"\
      -Label "Arrêt urgence activé SYSTEM OUT vers PLC" -DeviceMap "51"\
      -Category "PLC"

      -Name "SDO_MON_AutoOn" -SignalType "DO" -Device "DNet_Slave"\
      -Label "Mode Auto activé SYSTEM OUT vers PLC" -DeviceMap "52"\
      -Category "PLC"

      -Name "SDO_MON_RunChainOK" -SignalType "DO" -Device "DNet_Slave"\
      -Label "Chaîne sécurité OK SYSTEM OUT vers PLC" -DeviceMap "53"\
      -Category "PLC"

      -Name "SDO_MON_ExecError" -SignalType "DO" -Device "DNet_Slave"\
      -Label "Erreur exécution programme SYSTEM OUT vers PLC" -DeviceMap "54"\
      -Category "PLC"

      -Name "SDO_MON_MotorOnState" -SignalType "DO" -Device "DNet_Slave"\
      -Label "Moteurs activés SYSTEM OUT vers PLC" -DeviceMap "55"\
      -Category "PLC"

      -Name "SDO_MON_MotorOffState" -SignalType "DO" -Device "DNet_Slave"\
      -Label "Moteurs désactivés  SYSTEM OUT vers PLC" -DeviceMap "56"\
      -Category "PLC"

      -Name "SDO_MON_MotionSuprvTrig" -SignalType "DO" -Device "DNet_Slave"\
      -Label "Collision détecté SYSTEM OUT vers PLC" -DeviceMap "57"\
      -Category "PLC"

      -Name "SDO_MON_MotionSuprvOn" -SignalType "DO" -Device "DNet_Slave"\
      -Label "Supervision de collision activé SYSTEM OUT vers PLC"\
      -DeviceMap "58" -Category "PLC"

      -Name "SDO_MON_PathReturnErr" -SignalType "DO" -Device "DNet_Slave"\
      -Label "Erreur retour trajectoire SYSTEM OUT vers PLC" -DeviceMap "59"\
      -Category "PLC"

      -Name "SDO_MON_TaskExecMain" -SignalType "DO" -Device "DNet_Slave"\
      -Label "Tâche PRINCIPALE en ecécution SYSTEM OUT vers PLC" -DeviceMap "61"\
      -Category "PLC"

      -Name "SDO_PLCIN_14" -SignalType "DO" -Device "DNet_Slave"\
      -Label "SYSTEM OUT vers PLC via DNET" -DeviceMap "62" -Category "PLC"

      -Name "SAO_MON_TCPSpeed" -SignalType "AO" -Device "DNet_Slave"\
      -Label "Vitesse ROB_1" -DeviceMap "64-79" -Category "PLC"\
      -EncType "UNSIGNED" -MaxLog 10 -MaxBitVal 10000

      -Name "SDO_PLCIN_15" -SignalType "DO" -Device "DNet_Slave"\
      -Label "SYSTEM OUT vers PLC via DNET" -DeviceMap "63" -Category "PLC"

      -Name "DI_Virtuel1_Bouton1" -SignalType "DI" -Device "Virtuel"\
      -Label "Link to button 1" -DeviceMap "0" -Access "Local_AUTO"

      -Name "DI_Virtuel2_Bouton2" -SignalType "DI" -Device "Virtuel"\
      -Label "Link to button 2" -DeviceMap "1" -Access "Local_AUTO"

      -Name "DI_Virtuel3_Bouton3" -SignalType "DI" -Device "Virtuel"\
      -Label "Link to button 3" -DeviceMap "2" -Access "Local_AUTO"

      -Name "DI_Virtuel4_Bouton4" -SignalType "DI" -Device "Virtuel"\
      -Label "Link to button 4" -DeviceMap "3" -Access "Local_AUTO"

      -Name "DO_Virtuel1" -SignalType "DO" -Device "Virtuel"\
      -Label "Sortie virtuelle 1" -DeviceMap "0" -Access "Local_AUTO"

      -Name "DO_Virtuel2" -SignalType "DO" -Device "Virtuel"\
      -Label "Sortie virtuelle 2" -DeviceMap "1" -Access "Local_AUTO"

      -Name "DO_Virtuel3" -SignalType "DO" -Device "Virtuel"\
      -Label "Sortie virtuelle 3" -DeviceMap "2" -Access "Local_AUTO"

      -Name "DO_Virtuel4" -SignalType "DO" -Device "Virtuel"\
      -Label "Sortie virtuelle 4" -DeviceMap "3" -Access "Local_AUTO"

      -Name "SDI_ACT_StartAtCurrent_Cont" -SignalType "DI" -Device "DNet_Slave"\
      -Label "Exec au PP mode Cont SYSTEM IN du PLC" -DeviceMap "57"\
      -Category "PLC"

      -Name "SDI_ACT_StartAtMain_Cont" -SignalType "DI" -Device "DNet_Slave"\
      -Label "Exec PP to Main mode Cont SYSTEM IN du PLC" -DeviceMap "58"\
      -Category "PLC"

      -Name "AI_PLCOUT_01" -SignalType "AI" -Device "DNet_Slave"\
      -Label "AIN 01 (16bits) du PLC via DNET" -DeviceMap "96-111"\
      -Category "PLC" -MaxLog 1000 -MaxPhys 10000 -MaxBitVal 10000 -MinLog -1000\
      -MinPhys -10000 -MinBitVal -10000

      -Name "AI_PLCOUT_02" -SignalType "AI" -Device "DNet_Slave"\
      -Label "AIN 02 (16bits) du PLC via DNET" -DeviceMap "112-127"\
      -Category "PLC" -MaxLog 1000 -MaxPhys 10000 -MaxBitVal 10000 -MinLog -1000\
      -MinPhys -10000 -MinBitVal -10000

      -Name "AO_PLCIN_01" -SignalType "AO" -Device "DNet_Slave"\
      -Label "AO 01 (16bits) vers PLC via DNET" -DeviceMap "96-111"\
      -Category "PLC" -MaxLog 1000 -MaxPhys 10000 -MaxBitVal 10000 -MinLog -1000\
      -MinPhys -10000 -MinBitVal -10000

      -Name "AO_PLCIN_02" -SignalType "AO" -Device "DNet_Slave"\
      -Label "AO 02 (16bits) vers PLC via DNET" -DeviceMap "112-127"\
      -Category "PLC" -MaxLog 1000 -MaxPhys 10000 -MaxBitVal 10000 -MinLog -1000\
      -MinPhys -10000 -MinBitVal -10000

      -Name "AO_PLCIN_03" -SignalType "AO" -Device "DNet_Slave"\
      -Label "AO 03 (16bits) vers PLC via DNET" -DeviceMap "128-143"\
      -Category "PLC" -MaxLog 1000 -MaxPhys 10000 -MaxBitVal 10000 -MinLog -1000\
      -MinPhys -10000 -MinBitVal -10000

      -Name "AI_PLCOUT_03" -SignalType "AI" -Device "DNet_Slave"\
      -Label "AIN 03 (16bits) du PLC via DNET" -DeviceMap "128-143"\
      -Category "PLC" -MaxLog 1000 -MaxPhys 10000 -MaxBitVal 10000 -MinLog -1000\
      -MinPhys -10000 -MinBitVal -10000

      -Name "AI_PLCOUT_04" -SignalType "AI" -Device "DNet_Slave"\
      -Label "AIN 04 (16bits) du PLC via DNET" -DeviceMap "144-159"\
      -Category "PLC" -MaxLog 1000 -MaxPhys 10000 -MaxBitVal 10000 -MinLog -1000\
      -MinPhys -10000 -MinBitVal -10000

      -Name "AO_PLCIN_04" -SignalType "AO" -Device "DNet_Slave"\
      -Label "AO 04 (16bits) vers PLC via DNET" -DeviceMap "144-159"\
      -Category "PLC" -MaxLog 1000 -MaxPhys 10000 -MaxBitVal 10000 -MinLog -1000\
      -MinPhys -10000 -MinBitVal -10000

      -Name "DI_PLCOUT_16" -SignalType "DI" -Device "DNet_Slave"\
      -Label "DIN du PLC via DNET" -DeviceMap "80" -Category "PLC"

      -Name "DI_PLCOUT_17" -SignalType "DI" -Device "DNet_Slave"\
      -Label "DIN du PLC via DNET" -DeviceMap "81" -Category "PLC"

      -Name "DI_PLCOUT_18" -SignalType "DI" -Device "DNet_Slave"\
      -Label "DIN du PLC via DNET" -DeviceMap "82" -Category "PLC"

      -Name "DI_PLCOUT_19" -SignalType "DI" -Device "DNet_Slave"\
      -Label "DIN du PLC via DNET" -DeviceMap "83" -Category "PLC"

      -Name "DI_PLCOUT_20" -SignalType "DI" -Device "DNet_Slave"\
      -Label "DIN du PLC via DNET" -DeviceMap "84" -Category "PLC"

      -Name "DI_PLCOUT_21" -SignalType "DI" -Device "DNet_Slave"\
      -Label "DIN du PLC via DNET" -DeviceMap "85" -Category "PLC"

      -Name "DI_PLCOUT_22" -SignalType "DI" -Device "DNet_Slave"\
      -Label "DIN du PLC via DNET" -DeviceMap "86" -Category "PLC"

      -Name "DI_PLCOUT_23" -SignalType "DI" -Device "DNet_Slave"\
      -Label "DIN du PLC via DNET" -DeviceMap "87" -Category "PLC"

      -Name "DI_PLCOUT_24" -SignalType "DI" -Device "DNet_Slave"\
      -Label "DIN du PLC via DNET" -DeviceMap "88" -Category "PLC"

      -Name "DI_PLCOUT_25" -SignalType "DI" -Device "DNet_Slave"\
      -Label "DIN du PLC via DNET" -DeviceMap "89" -Category "PLC"

      -Name "DI_PLCOUT_26" -SignalType "DI" -Device "DNet_Slave"\
      -Label "DIN du PLC via DNET" -DeviceMap "90" -Category "PLC"

      -Name "DI_PLCOUT_27" -SignalType "DI" -Device "DNet_Slave"\
      -Label "DIN du PLC via DNET" -DeviceMap "91" -Category "PLC"

      -Name "DI_PLCOUT_28" -SignalType "DI" -Device "DNet_Slave"\
      -Label "DIN du PLC via DNET" -DeviceMap "92" -Category "PLC"

      -Name "DI_PLCOUT_29" -SignalType "DI" -Device "DNet_Slave"\
      -Label "DIN du PLC via DNET" -DeviceMap "93" -Category "PLC"

      -Name "DI_PLCOUT_30" -SignalType "DI" -Device "DNet_Slave"\
      -Label "DIN du PLC via DNET" -DeviceMap "94" -Category "PLC"

      -Name "DI_PLCOUT_31" -SignalType "DI" -Device "DNet_Slave"\
      -Label "DIN du PLC via DNET" -DeviceMap "95" -Category "PLC"

      -Name "DO_PLCIN_16" -SignalType "DO" -Device "DNet_Slave"\
      -Label "DOUT vers PLC via DNET" -DeviceMap "80" -Category "PLC"

      -Name "DO_PLCIN_17" -SignalType "DO" -Device "DNet_Slave"\
      -Label "DOUT vers PLC via DNET" -DeviceMap "81" -Category "PLC"

      -Name "DO_PLCIN_18" -SignalType "DO" -Device "DNet_Slave"\
      -Label "DOUT vers PLC via DNET" -DeviceMap "82" -Category "PLC"

      -Name "DO_PLCIN_19" -SignalType "DO" -Device "DNet_Slave"\
      -Label "DOUT vers PLC via DNET" -DeviceMap "83" -Category "PLC"

      -Name "DO_PLCIN_20" -SignalType "DO" -Device "DNet_Slave"\
      -Label "DOUT vers PLC via DNET" -DeviceMap "84" -Category "PLC"

      -Name "DO_PLCIN_21" -SignalType "DO" -Device "DNet_Slave"\
      -Label "DOUT vers PLC via DNET" -DeviceMap "85" -Category "PLC"

      -Name "DO_PLCIN_22" -SignalType "DO" -Device "DNet_Slave"\
      -Label "DOUT vers PLC via DNET" -DeviceMap "86" -Category "PLC"

      -Name "DO_PLCIN_23" -SignalType "DO" -Device "DNet_Slave"\
      -Label "DOUT vers PLC via DNET" -DeviceMap "87" -Category "PLC"

      -Name "DO_PLCIN_24" -SignalType "DO" -Device "DNet_Slave"\
      -Label "DOUT vers PLC via DNET" -DeviceMap "88" -Category "PLC"

      -Name "DO_PLCIN_25" -SignalType "DO" -Device "DNet_Slave"\
      -Label "DOUT vers PLC via DNET" -DeviceMap "89" -Category "PLC"

      -Name "DO_PLCIN_26" -SignalType "DO" -Device "DNet_Slave"\
      -Label "DOUT vers PLC via DNET" -DeviceMap "90" -Category "PLC"

      -Name "DO_PLCIN_27" -SignalType "DO" -Device "DNet_Slave"\
      -Label "DOUT vers PLC via DNET" -DeviceMap "91" -Category "PLC"

      -Name "DO_PLCIN_28" -SignalType "DO" -Device "DNet_Slave"\
      -Label "DOUT vers PLC via DNET" -DeviceMap "92" -Category "PLC"

      -Name "DO_PLCIN_29" -SignalType "DO" -Device "DNet_Slave"\
      -Label "DOUT vers PLC via DNET" -DeviceMap "93" -Category "PLC"

      -Name "DO_PLCIN_30" -SignalType "DO" -Device "DNet_Slave"\
      -Label "DOUT vers PLC via DNET" -DeviceMap "94" -Category "PLC"

      -Name "DO_PLCIN_31" -SignalType "DO" -Device "DNet_Slave"\
      -Label "DOUT vers PLC via DNET" -DeviceMap "95" -Category "PLC"

      -Name "DI_Virtuel5" -SignalType "DI" -Device "Virtuel"\
      -Label "Entrée virtuelle 5" -DeviceMap "4" -Access "Local_AUTO"

      -Name "DI_Virtuel6" -SignalType "DI" -Device "Virtuel"\
      -Label "Entrée virtuelle 6" -DeviceMap "5" -Access "Local_AUTO"

      -Name "DI_Virtuel7" -SignalType "DI" -Device "Virtuel"\
      -Label "Entrée virtuelle 7" -DeviceMap "6" -Access "Local_AUTO"

      -Name "DI_Virtuel8" -SignalType "DI" -Device "Virtuel"\
      -Label "Entrée virtuelle 8" -DeviceMap "7" -Access "Local_AUTO"
